LIN {X 0,Y 573.063,Z 619.264,A -85,B 0,C 180,E1 -2090.645,E2 -2090.645} C_VEL
LIN {X 0,Y 573.121,Z 612.909,A -85,B 0,C 180,E1 -2091.584,E2 -2091.584} C_VEL
LIN {X 0,Y 573.201,Z 605.158,A -85,B 0,C 180,E1 -2092.528,E2 -2092.528} C_VEL
LIN {X 0,Y 573.3,Z 596.066,A -85,B 0,C 180,E1 -2093.44,E2 -2093.44} C_VEL
LIN {X 0,Y 573.417,Z 584.971,A -85,B 0,C 180,E1 -2094.337,E2 -2094.337} C_VEL
LIN {X 0,Y 573.555,Z 572.942,A -85,B 0,C 180,E1 -2095.095,E2 -2095.095} C_VEL
LIN {X 0,Y 573.613,Z 562.036,A -85,B 0,C 180,E1 -2095.635,E2 -2095.635} C_VEL
LIN {X 0,Y 573.65,Z 554.886,A -85,B 0,C 180,E1 -2095.926,E2 -2095.926} C_VEL
LIN {X 0,Y 573.305,Z 553.075,A -85,B 0,C 180,E1 -2096.016,E2 -2096.016} C_VEL
LIN {X 0,Y 573.234,Z 553.082,A -85,B 0,C 180,E1 -2098.564,E2 -2098.564} C_VEL
LIN {X 0,Y 573.238,Z 553.081,A -85,B 0,C 180,E1 -2100.992,E2 -2100.992} C_VEL
LIN {X 0,Y 573.256,Z 553.079,A -85,B 0,C 180,E1 -2103.523,E2 -2103.523} C_VEL
LIN {X 0,Y 573.239,Z 553.082,A -85,B 0,C 180,E1 -2106.049,E2 -2106.049} C_VEL
LIN {X 0,Y 573.245,Z 553.083,A -85,B 0,C 180,E1 -2108.7,E2 -2108.7} C_VEL
LIN {X 0,Y 573.305,Z 553.158,A -85,B 0,C 180,E1 -2111.493,E2 -2111.493} C_VEL
LIN {X 0,Y 573.377,Z 559.685,A -85,B 0,C 180,E1 -2113.683,E2 -2113.683} C_VEL
LIN {X 0,Y 573.399,Z 567.264,A -85,B 0,C 180,E1 -2116.313,E2 -2116.313} C_VEL
LIN {X 0,Y 573.383,Z 575.18,A -85,B 0,C 180,E1 -2119.024,E2 -2119.024} C_VEL
LIN {X 0,Y 573.289,Z 582.833,A -85,B 0,C 180,E1 -2121.68,E2 -2121.68} C_VEL
LIN {X 0,Y 573.249,Z 590.784,A -85,B 0,C 180,E1 -2124.414,E2 -2124.414} C_VEL
LIN {X 0,Y 573.184,Z 599.505,A -85,B 0,C 180,E1 -2127.351,E2 -2127.351} C_VEL
LIN {X 0,Y 573.114,Z 608.136,A -85,B 0,C 180,E1 -2130.206,E2 -2130.206} C_VEL
LIN {X 0,Y 573.085,Z 615.536,A -85,B 0,C 180,E1 -2132.621,E2 -2132.621} C_VEL
LIN {X 0,Y 573.073,Z 621.489,A -85,B 0,C 180,E1 -2134.545,E2 -2134.545} C_VEL
LIN {X 0,Y 573.86,Z 627.22,A -85,B 0,C 180,E1 -2134.666,E2 -2134.666} C_VEL
LIN {X 0,Y 573.753,Z 640.519,A -85,B 0,C 180,E1 -2135.015,E2 -2135.015} C_VEL
LIN {X 0,Y 573.656,Z 652.623,A -85,B 0,C 180,E1 -2135.48,E2 -2135.48} C_VEL
LIN {X 0,Y 573.494,Z 663.949,A -85,B 0,C 180,E1 -2136.05,E2 -2136.05} C_VEL
LIN {X 0,Y 573.407,Z 674.306,A -85,B 0,C 180,E1 -2136.708,E2 -2136.708} C_VEL
LIN {X 0,Y 573.316,Z 685.226,A -85,B 0,C 180,E1 -2137.571,E2 -2137.571} C_VEL
LIN {X 0,Y 573.206,Z 693.9,A -85,B 0,C 180,E1 -2138.419,E2 -2138.419} C_VEL
LIN {X 0,Y 573.133,Z 701.824,A -85,B 0,C 180,E1 -2139.357,E2 -2139.357} C_VEL
LIN {X 0,Y 573.082,Z 708.329,A -85,B 0,C 180,E1 -2140.291,E2 -2140.291} C_VEL
LIN {X 0,Y 573.063,Z 714.612,A -85,B 0,C 180,E1 -2141.406,E2 -2141.406} C_VEL
LIN {X 0,Y 572.981,Z 719.505,A -85,B 0,C 180,E1 -2142.512,E2 -2142.512} C_VEL
LIN {X 0,Y 572.958,Z 723.194,A -85,B 0,C 180,E1 -2143.613,E2 -2143.613} C_VEL
LIN {X 0,Y 572.955,Z 725.025,A -85,B 0,C 180,E1 -2144.345,E2 -2144.345} C_VEL
LIN {X 0,Y 572.968,Z 727.243,A -85,B 0,C 180,E1 -2145.694,E2 -2145.694} C_VEL
LIN {X 0,Y 572.962,Z 727.858,A -85,B 0,C 180,E1 -2146.523,E2 -2146.523} C_VEL
LIN {X 0,Y 572.941,Z 727.962,A -85,B 0,C 180,E1 -2147.244,E2 -2147.244} C_VEL
LIN {X 0,Y 572.94,Z 727.643,A -85,B 0,C 180,E1 -2147.964,E2 -2147.964} C_VEL
LIN {X 0,Y 573.025,Z 726.662,A -85,B 0,C 180,E1 -2148.86,E2 -2148.86} C_VEL
LIN {X 0,Y 572.976,Z 724.178,A -85,B 0,C 180,E1 -2150.112,E2 -2150.112} C_VEL
LIN {X 0,Y 572.998,Z 720.982,A -85,B 0,C 180,E1 -2151.181,E2 -2151.181} C_VEL
LIN {X 0,Y 573.046,Z 716.722,A -85,B 0,C 180,E1 -2152.247,E2 -2152.247} C_VEL
LIN {X 0,Y 573.054,Z 710.771,A -85,B 0,C 180,E1 -2153.4,E2 -2153.4} C_VEL
LIN {X 0,Y 573.09,Z 704.512,A -85,B 0,C 180,E1 -2154.37,E2 -2154.37} C_VEL
LIN {X 0,Y 573.163,Z 697.624,A -85,B 0,C 180,E1 -2155.253,E2 -2155.253} C_VEL
LIN {X 0,Y 573.268,Z 689.333,A -85,B 0,C 180,E1 -2156.134,E2 -2156.134} C_VEL
LIN {X 0,Y 573.399,Z 680.335,A -85,B 0,C 180,E1 -2156.926,E2 -2156.926} C_VEL
LIN {X 0,Y 573.463,Z 669.337,A -85,B 0,C 180,E1 -2157.718,E2 -2157.718} C_VEL
LIN {X 0,Y 573.596,Z 656.798,A -85,B 0,C 180,E1 -2158.421,E2 -2158.421} C_VEL
LIN {X 0,Y 573.721,Z 645.415,A -85,B 0,C 180,E1 -2158.904,E2 -2158.904} C_VEL
LIN {X 0,Y 573.801,Z 633.497,A -85,B 0,C 180,E1 -2159.277,E2 -2159.277} C_VEL
LIN {X 0,Y 573.603,Z 624.918,A -85,B 0,C 180,E1 -2159.474,E2 -2159.474} C_VEL
LIN {X 0,Y 573.104,Z 621.456,A -85,B 0,C 180,E1 -2159.561,E2 -2159.561} C_VEL
LIN {X 0,Y 573.138,Z 612.541,A -85,B 0,C 180,E1 -2162.46,E2 -2162.46} C_VEL
LIN {X 0,Y 573.174,Z 603.996,A -85,B 0,C 180,E1 -2165.277,E2 -2165.277} C_VEL
LIN {X 0,Y 573.213,Z 595.549,A -85,B 0,C 180,E1 -2168.106,E2 -2168.106} C_VEL
LIN {X 0,Y 573.281,Z 588.239,A -85,B 0,C 180,E1 -2170.597,E2 -2170.597} C_VEL
LIN {X 0,Y 573.32,Z 579.984,A -85,B 0,C 180,E1 -2173.469,E2 -2173.469} C_VEL
LIN {X 0,Y 573.365,Z 573.728,A -85,B 0,C 180,E1 -2175.645,E2 -2175.645} C_VEL
LIN {X 0,Y 573.328,Z 565.652,A -85,B 0,C 180,E1 -2178.215,E2 -2178.215} C_VEL
LIN {X 0,Y 573.17,Z 557.031,A -85,B 0,C 180,E1 -2180.83,E2 -2180.83} C_VEL
LIN {X 0,Y 573.181,Z 553.092,A -85,B 0,C 180,E1 -2181.961,E2 -2181.961} C_VEL
LIN {X 0,Y 573.264,Z 553.082,A -85,B 0,C 180,E1 -2184.88,E2 -2184.88} C_VEL
LIN {X 0,Y 573.284,Z 553.077,A -85,B 0,C 180,E1 -2187.765,E2 -2187.765} C_VEL
LIN {X 0,Y 573.253,Z 553.083,A -85,B 0,C 180,E1 -2190.176,E2 -2190.176} C_VEL
LIN {X 0,Y 573.253,Z 553.08,A -85,B 0,C 180,E1 -2192.645,E2 -2192.645} C_VEL
LIN {X 0,Y 573.265,Z 553.08,A -85,B 0,C 180,E1 -2195.184,E2 -2195.184} C_VEL
LIN {X 0,Y 573.232,Z 553.083,A -85,B 0,C 180,E1 -2197.808,E2 -2197.808} C_VEL
LIN {X 0,Y 573.265,Z 553.081,A -85,B 0,C 180,E1 -2200.529,E2 -2200.529} C_VEL
LIN {X 0,Y 573.248,Z 553.083,A -85,B 0,C 180,E1 -2203.671,E2 -2203.671} C_VEL
LIN {X 0,Y 573.244,Z 553.083,A -85,B 0,C 180,E1 -2206.643,E2 -2206.643} C_VEL
LIN {X 0,Y 573.271,Z 553.079,A -85,B 0,C 180,E1 -2209.478,E2 -2209.478} C_VEL
LIN {X 0,Y 573.236,Z 553.084,A -85,B 0,C 180,E1 -2212.194,E2 -2212.194} C_VEL
LIN {X 0,Y 573.29,Z 553.151,A -85,B 0,C 180,E1 -2213.301,E2 -2213.301} C_VEL
LIN {X 0,Y 574.101,Z 558.468,A -85,B 0,C 180,E1 -2214.446,E2 -2214.446} C_VEL
LIN {X 0,Y 574.123,Z 573.3,A -85,B 0,C 180,E1 -2217.412,E2 -2217.412} C_VEL
LIN {X 0,Y 574.135,Z 587.619,A -85,B 0,C 180,E1 -2220.163,E2 -2220.163} C_VEL
LIN {X 0,Y 574.037,Z 598.461,A -85,B 0,C 180,E1 -2222.275,E2 -2222.275} C_VEL
LIN {X 0,Y 573.854,Z 614.175,A -85,B 0,C 180,E1 -2225.394,E2 -2225.394} C_VEL
LIN {X 0,Y 573.637,Z 629.889,A -85,B 0,C 180,E1 -2228.436,E2 -2228.436} C_VEL
LIN {X 0,Y 573.459,Z 645.603,A -85,B 0,C 180,E1 -2231.42,E2 -2231.42} C_VEL
LIN {X 0,Y 573.327,Z 659.353,A -85,B 0,C 180,E1 -2233.99,E2 -2233.99} C_VEL
LIN {X 0,Y 573.205,Z 675.067,A -85,B 0,C 180,E1 -2236.89,E2 -2236.89} C_VEL
LIN {X 0,Y 573.204,Z 678.139,A -85,B 0,C 180,E1 -2237.453,E2 -2237.453} C_VEL
LIN {X 0,Y 573.867,Z 683.985,A -85,B 0,C 180,E1 -2237.558,E2 -2237.558} C_VEL
LIN {X 0,Y 573.787,Z 697.245,A -85,B 0,C 180,E1 -2237.87,E2 -2237.87} C_VEL
LIN {X 0,Y 573.713,Z 709.391,A -85,B 0,C 180,E1 -2238.295,E2 -2238.295} C_VEL
LIN {X 0,Y 573.573,Z 720.61,A -85,B 0,C 180,E1 -2238.818,E2 -2238.818} C_VEL
LIN {X 0,Y 573.471,Z 731.924,A -85,B 0,C 180,E1 -2239.497,E2 -2239.497} C_VEL
LIN {X 0,Y 573.351,Z 742.548,A -85,B 0,C 180,E1 -2240.298,E2 -2240.298} C_VEL
LIN {X 0,Y 573.24,Z 752.12,A -85,B 0,C 180,E1 -2241.185,E2 -2241.185} C_VEL
LIN {X 0,Y 573.16,Z 759.966,A -85,B 0,C 180,E1 -2242.072,E2 -2242.072} C_VEL
LIN {X 0,Y 573.072,Z 767.958,A -85,B 0,C 180,E1 -2243.186,E2 -2243.186} C_VEL
LIN {X 0,Y 573.07,Z 774.684,A -85,B 0,C 180,E1 -2244.37,E2 -2244.37} C_VEL
LIN {X 0,Y 573.029,Z 779.374,A -85,B 0,C 180,E1 -2245.428,E2 -2245.428} C_VEL
LIN {X 0,Y 573.022,Z 782.959,A -85,B 0,C 180,E1 -2246.485,E2 -2246.485} C_VEL
LIN {X 0,Y 572.959,Z 784.81,A -85,B 0,C 180,E1 -2247.188,E2 -2247.188} C_VEL
LIN {X 0,Y 572.937,Z 786.201,A -85,B 0,C 180,E1 -2247.892,E2 -2247.892} C_VEL
LIN {X 0,Y 572.94,Z 787.785,A -85,B 0,C 180,E1 -2249.298,E2 -2249.298} C_VEL
LIN {X 0,Y 572.938,Z 788,A -85,B 0,C 180,E1 -2250.001,E2 -2250.001} C_VEL
LIN {X 0,Y 572.946,Z 787.185,A -85,B 0,C 180,E1 -2251.406,E2 -2251.406} C_VEL
LIN {X 0,Y 572.937,Z 786.199,A -85,B 0,C 180,E1 -2252.11,E2 -2252.11} C_VEL
LIN {X 0,Y 572.959,Z 784.808,A -85,B 0,C 180,E1 -2252.813,E2 -2252.813} C_VEL
LIN {X 0,Y 573.014,Z 781.894,A -85,B 0,C 180,E1 -2253.869,E2 -2253.869} C_VEL
LIN {X 0,Y 572.963,Z 777.947,A -85,B 0,C 180,E1 -2254.926,E2 -2254.926} C_VEL
LIN {X 0,Y 573.064,Z 771.874,A -85,B 0,C 180,E1 -2256.161,E2 -2256.161} C_VEL
LIN {X 0,Y 573.12,Z 765.233,A -85,B 0,C 180,E1 -2257.221,E2 -2257.221} C_VEL
LIN {X 0,Y 573.199,Z 756.985,A -85,B 0,C 180,E1 -2258.284,E2 -2258.284} C_VEL
LIN {X 0,Y 573.287,Z 748.532,A -85,B 0,C 180,E1 -2259.171,E2 -2259.171} C_VEL
LIN {X 0,Y 573.42,Z 738.089,A -85,B 0,C 180,E1 -2260.059,E2 -2260.059} C_VEL
LIN {X 0,Y 573.554,Z 726.423,A -85,B 0,C 180,E1 -2260.853,E2 -2260.853} C_VEL
LIN {X 0,Y 573.618,Z 714.869,A -85,B 0,C 180,E1 -2261.467,E2 -2261.467} C_VEL
LIN {X 0,Y 573.731,Z 702.158,A -85,B 0,C 180,E1 -2261.975,E2 -2261.975} C_VEL
LIN {X 0,Y 573.855,Z 689.497,A -85,B 0,C 180,E1 -2262.331,E2 -2262.331} C_VEL
LIN {X 0,Y 573.668,Z 681.259,A -85,B 0,C 180,E1 -2262.49,E2 -2262.49} C_VEL
LIN {X 0,Y 573.194,Z 678.031,A -85,B 0,C 180,E1 -2262.571,E2 -2262.571} C_VEL
LIN {X 0,Y 573.319,Z 663.358,A -85,B 0,C 180,E1 -2265.282,E2 -2265.282} C_VEL
LIN {X 0,Y 573.458,Z 647.707,A -85,B 0,C 180,E1 -2268.211,E2 -2268.211} C_VEL
LIN {X 0,Y 573.616,Z 632.538,A -85,B 0,C 180,E1 -2271.096,E2 -2271.096} C_VEL
LIN {X 0,Y 573.768,Z 618.361,A -85,B 0,C 180,E1 -2273.842,E2 -2273.842} C_VEL
LIN {X 0,Y 573.962,Z 604.222,A -85,B 0,C 180,E1 -2276.637,E2 -2276.637} C_VEL
LIN {X 0,Y 574.103,Z 590.754,A -85,B 0,C 180,E1 -2279.319,E2 -2279.319} C_VEL
LIN {X 0,Y 574.085,Z 576.51,A -85,B 0,C 180,E1 -2282.063,E2 -2282.063} C_VEL
LIN {X 0,Y 574.126,Z 563.882,A -85,B 0,C 180,E1 -2284.583,E2 -2284.583} C_VEL
LIN {X 0,Y 573.987,Z 556.687,A -85,B 0,C 180,E1 -2286.087,E2 -2286.087} C_VEL
LIN {X 0,Y 573.258,Z 553.081,A -85,B 0,C 180,E1 -2286.922,E2 -2286.922} C_VEL
LIN {X 0,Y 573.253,Z 553.082,A -85,B 0,C 180,E1 -2289.607,E2 -2289.607} C_VEL
LIN {X 0,Y 573.245,Z 553.08,A -85,B 0,C 180,E1 -2292.642,E2 -2292.642} C_VEL
LIN {X 0,Y 573.237,Z 553.084,A -85,B 0,C 180,E1 -2295.666,E2 -2295.666} C_VEL
LIN {X 0,Y 573.243,Z 553.081,A -85,B 0,C 180,E1 -2298.544,E2 -2298.544} C_VEL
LIN {X 0,Y 573.243,Z 553.082,A -85,B 0,C 180,E1 -2301.298,E2 -2301.298} C_VEL
LIN {X 0,Y 573.27,Z 553.079,A -85,B 0,C 180,E1 -2304.011,E2 -2304.011} C_VEL
LIN {X 0,Y 573.274,Z 553.077,A -85,B 0,C 180,E1 -2306.518,E2 -2306.518} C_VEL
LIN {X 0,Y 573.232,Z 553.082,A -85,B 0,C 180,E1 -2309.118,E2 -2309.118} C_VEL
LIN {X 0,Y 573.268,Z 553.08,A -85,B 0,C 180,E1 -2311.969,E2 -2311.969} C_VEL
LIN {X 0,Y 573.259,Z 553.079,A -85,B 0,C 180,E1 -2314.59,E2 -2314.59} C_VEL
LIN {X 0,Y 573.241,Z 553.082,A -85,B 0,C 180,E1 -2317.662,E2 -2317.662} C_VEL
LIN {X 0,Y 573.283,Z 553.076,A -85,B 0,C 180,E1 -2320.728,E2 -2320.728} C_VEL
LIN {X 0,Y 573.256,Z 553.081,A -85,B 0,C 180,E1 -2323.622,E2 -2323.622} C_VEL
LIN {X 0,Y 573.277,Z 553.077,A -85,B 0,C 180,E1 -2325.807,E2 -2325.807} C_VEL
LIN {X 0,Y 573.267,Z 553.078,A -85,B 0,C 180,E1 -2328.745,E2 -2328.745} C_VEL
LIN {X 0,Y 573.293,Z 553.075,A -85,B 0,C 180,E1 -2331.54,E2 -2331.54} C_VEL
LIN {X 0,Y 573.294,Z 553.076,A -85,B 0,C 180,E1 -2334.372,E2 -2334.372} C_VEL
LIN {X 0,Y 573.306,Z 553.074,A -85,B 0,C 180,E1 -2337.892,E2 -2337.892} C_VEL
LIN {X 0,Y 573.336,Z 553.069,A -85,B 0,C 180,E1 -2340.702,E2 -2340.702} C_VEL
LIN {X 0,Y 573.233,Z 553.084,A -85,B 0,C 180,E1 -2343.514,E2 -2343.514} C_VEL
LIN {X 0,Y 573.293,Z 553.075,A -85,B 0,C 180,E1 -2345.628,E2 -2345.628} C_VEL
LIN {X 0,Y 573.288,Z 553.076,A -85,B 0,C 180,E1 -2348.459,E2 -2348.459} C_VEL
LIN {X 0,Y 573.275,Z 553.077,A -85,B 0,C 180,E1 -2351.312,E2 -2351.312} C_VEL
LIN {X 0,Y 573.277,Z 553.078,A -85,B 0,C 180,E1 -2354.193,E2 -2354.193} C_VEL
LIN {X 0,Y 573.261,Z 553.079,A -85,B 0,C 180,E1 -2357.111,E2 -2357.111} C_VEL
LIN {X 0,Y 573.254,Z 553.081,A -85,B 0,C 180,E1 -2360.076,E2 -2360.076} C_VEL
LIN {X 0,Y 573.237,Z 553.082,A -85,B 0,C 180,E1 -2363.099,E2 -2363.099} C_VEL
LIN {X 0,Y 573.252,Z 553.079,A -85,B 0,C 180,E1 -2364.389,E2 -2364.389} C_VEL
LIN {X 0,Y 572.624,Z 553.16,A -85,B 0,C 180,E1 -2364.975,E2 -2364.975} C_VEL
LIN {X 0,Y 569.777,Z 553.515,A -85,B 0,C 180,E1 -2365.927,E2 -2365.927} C_VEL
LIN {X 0,Y 567.345,Z 553.817,A -85,B 0,C 180,E1 -2366.692,E2 -2366.692} C_VEL
LIN {X 0,Y 566.295,Z 553.945,A -85,B 0,C 180,E1 -2367.283,E2 -2367.283} C_VEL
LIN {X 0,Y 566.209,Z 553.956,A -85,B 0,C 180,E1 -2367.483,E2 -2367.483} C_VEL
LIN {X 0,Y 566.203,Z 553.957,A -85,B 0,C 180,E1 -2369.768,E2 -2369.768} C_VEL
LIN {X 0,Y 566.205,Z 553.958,A -85,B 0,C 180,E1 -2372.43,E2 -2372.43} C_VEL
LIN {X 0,Y 566.214,Z 553.959,A -85,B 0,C 180,E1 -2374.994,E2 -2374.994} C_VEL
LIN {X 0,Y 566.198,Z 553.96,A -85,B 0,C 180,E1 -2377.46,E2 -2377.46} C_VEL
LIN {X 0,Y 566.219,Z 553.956,A -85,B 0,C 180,E1 -2380.198,E2 -2380.198} C_VEL
LIN {X 0,Y 566.206,Z 553.959,A -85,B 0,C 180,E1 -2383.053,E2 -2383.053} C_VEL
LIN {X 0,Y 566.203,Z 553.958,A -85,B 0,C 180,E1 -2386.048,E2 -2386.048} C_VEL
LIN {X 0,Y 566.213,Z 553.958,A -85,B 0,C 180,E1 -2388.863,E2 -2388.863} C_VEL
LIN {X 0,Y 566.191,Z 553.96,A -85,B 0,C 180,E1 -2391.637,E2 -2391.637} C_VEL
LIN {X 0,Y 566.163,Z 553.963,A -85,B 0,C 180,E1 -2394.307,E2 -2394.307} C_VEL
LIN {X 0,Y 566.222,Z 553.956,A -85,B 0,C 180,E1 -2396.897,E2 -2396.897} C_VEL
LIN {X 0,Y 566.19,Z 553.961,A -85,B 0,C 180,E1 -2399.407,E2 -2399.407} C_VEL
LIN {X 0,Y 566.212,Z 553.958,A -85,B 0,C 180,E1 -2401.857,E2 -2401.857} C_VEL
LIN {X 0,Y 566.217,Z 553.959,A -85,B 0,C 180,E1 -2404.251,E2 -2404.251} C_VEL
LIN {X 0,Y 566.193,Z 553.961,A -85,B 0,C 180,E1 -2406.713,E2 -2406.713} C_VEL
LIN {X 0,Y 566.213,Z 553.956,A -85,B 0,C 180,E1 -2409.662,E2 -2409.662} C_VEL
LIN {X 0,Y 566.2,Z 553.959,A -85,B 0,C 180,E1 -2412.668,E2 -2412.668} C_VEL
LIN {X 0,Y 566.234,Z 553.954,A -85,B 0,C 180,E1 -2415.626,E2 -2415.626} C_VEL
LIN {X 0,Y 566.235,Z 553.954,A -85,B 0,C 180,E1 -2418.674,E2 -2418.674} C_VEL
LIN {X 0,Y 566.228,Z 553.955,A -85,B 0,C 180,E1 -2421.434,E2 -2421.434} C_VEL
LIN {X 0,Y 566.259,Z 553.952,A -85,B 0,C 180,E1 -2424.301,E2 -2424.301} C_VEL
LIN {X 0,Y 566.284,Z 553.949,A -85,B 0,C 180,E1 -2427.866,E2 -2427.866} C_VEL
LIN {X 0,Y 566.299,Z 553.946,A -85,B 0,C 180,E1 -2430.71,E2 -2430.71} C_VEL
LIN {X 0,Y 566.275,Z 554.004,A -85,B 0,C 180,E1 -2431.977,E2 -2431.977} C_VEL
LIN {X 0,Y 566.733,Z 557.867,A -85,B 0,C 180,E1 -2432.131,E2 -2432.131} C_VEL
LIN {X 0,Y 566.607,Z 569.41,A -85,B 0,C 180,E1 -2432.665,E2 -2432.665} C_VEL
LIN {X 0,Y 566.525,Z 578.649,A -85,B 0,C 180,E1 -2433.199,E2 -2433.199} C_VEL
LIN {X 0,Y 566.351,Z 588.706,A -85,B 0,C 180,E1 -2433.913,E2 -2433.913} C_VEL
LIN {X 0,Y 566.246,Z 597.047,A -85,B 0,C 180,E1 -2434.627,E2 -2434.627} C_VEL
LIN {X 0,Y 566.182,Z 604.132,A -85,B 0,C 180,E1 -2435.341,E2 -2435.341} C_VEL
LIN {X 0,Y 566.126,Z 611.583,A -85,B 0,C 180,E1 -2436.235,E2 -2436.235} C_VEL
LIN {X 0,Y 566.053,Z 617.821,A -85,B 0,C 180,E1 -2437.131,E2 -2437.131} C_VEL
LIN {X 0,Y 565.982,Z 622.123,A -85,B 0,C 180,E1 -2437.85,E2 -2437.85} C_VEL
LIN {X 0,Y 565.941,Z 627.374,A -85,B 0,C 180,E1 -2438.929,E2 -2438.929} C_VEL
LIN {X 0,Y 565.925,Z 631.479,A -85,B 0,C 180,E1 -2440.012,E2 -2440.012} C_VEL
LIN {X 0,Y 565.882,Z 634.643,A -85,B 0,C 180,E1 -2441.146,E2 -2441.146} C_VEL
LIN {X 0,Y 565.863,Z 636.61,A -85,B 0,C 180,E1 -2442.188,E2 -2442.188} C_VEL
LIN {X 0,Y 565.842,Z 637.503,A -85,B 0,C 180,E1 -2442.918,E2 -2442.918} C_VEL
LIN {X 0,Y 565.872,Z 637.914,A -85,B 0,C 180,E1 -2444.382,E2 -2444.382} C_VEL
LIN {X 0,Y 565.809,Z 637.547,A -85,B 0,C 180,E1 -2445.119,E2 -2445.119} C_VEL
LIN {X 0,Y 565.87,Z 635.393,A -85,B 0,C 180,E1 -2446.597,E2 -2446.597} C_VEL
LIN {X 0,Y 565.898,Z 632.603,A -85,B 0,C 180,E1 -2447.713,E2 -2447.713} C_VEL
LIN {X 0,Y 565.905,Z 628.683,A -85,B 0,C 180,E1 -2448.837,E2 -2448.837} C_VEL
LIN {X 0,Y 565.965,Z 625.43,A -85,B 0,C 180,E1 -2449.589,E2 -2449.589} C_VEL
LIN {X 0,Y 566,Z 619.275,A -85,B 0,C 180,E1 -2450.724,E2 -2450.724} C_VEL
LIN {X 0,Y 566.078,Z 612.656,A -85,B 0,C 180,E1 -2451.711,E2 -2451.711} C_VEL
LIN {X 0,Y 566.15,Z 605.171,A -85,B 0,C 180,E1 -2452.632,E2 -2452.632} C_VEL
LIN {X 0,Y 566.26,Z 596.693,A -85,B 0,C 180,E1 -2453.497,E2 -2453.497} C_VEL
LIN {X 0,Y 566.375,Z 586.308,A -85,B 0,C 180,E1 -2454.367,E2 -2454.367} C_VEL
LIN {X 0,Y 566.561,Z 575.227,A -85,B 0,C 180,E1 -2455.105,E2 -2455.105} C_VEL
LIN {X 0,Y 566.628,Z 563.2,A -85,B 0,C 180,E1 -2455.728,E2 -2455.728} C_VEL
LIN {X 0,Y 566.545,Z 555.337,A -85,B 0,C 180,E1 -2456.061,E2 -2456.061} C_VEL
LIN {X 0,Y 566.248,Z 553.953,A -85,B 0,C 180,E1 -2456.117,E2 -2456.117} C_VEL
LIN {X 0,Y 566.19,Z 553.96,A -85,B 0,C 180,E1 -2458.952,E2 -2458.952} C_VEL
LIN {X 0,Y 566.2,Z 553.959,A -85,B 0,C 180,E1 -2461.42,E2 -2461.42} C_VEL
LIN {X 0,Y 566.204,Z 553.959,A -85,B 0,C 180,E1 -2463.955,E2 -2463.955} C_VEL
LIN {X 0,Y 566.205,Z 553.958,A -85,B 0,C 180,E1 -2466.568,E2 -2466.568} C_VEL
LIN {X 0,Y 566.21,Z 553.959,A -85,B 0,C 180,E1 -2469.686,E2 -2469.686} C_VEL
LIN {X 0,Y 566.259,Z 554.067,A -85,B 0,C 180,E1 -2471.427,E2 -2471.427} C_VEL
LIN {X 0,Y 566.367,Z 561.664,A -85,B 0,C 180,E1 -2474.018,E2 -2474.018} C_VEL
LIN {X 0,Y 566.354,Z 570.107,A -85,B 0,C 180,E1 -2476.961,E2 -2476.961} C_VEL
LIN {X 0,Y 566.313,Z 578.345,A -85,B 0,C 180,E1 -2479.81,E2 -2479.81} C_VEL
LIN {X 0,Y 566.246,Z 586.39,A -85,B 0,C 180,E1 -2482.591,E2 -2482.591} C_VEL
LIN {X 0,Y 566.192,Z 593.88,A -85,B 0,C 180,E1 -2485.181,E2 -2485.181} C_VEL
LIN {X 0,Y 566.104,Z 602.65,A -85,B 0,C 180,E1 -2488.155,E2 -2488.155} C_VEL
LIN {X 0,Y 566.055,Z 610.261,A -85,B 0,C 180,E1 -2490.695,E2 -2490.695} C_VEL
LIN {X 0,Y 566.004,Z 618.62,A -85,B 0,C 180,E1 -2493.448,E2 -2493.448} C_VEL
LIN {X 0,Y 566.002,Z 621.485,A -85,B 0,C 180,E1 -2494.385,E2 -2494.385} C_VEL
LIN {X 0,Y 566.933,Z 628.252,A -85,B 0,C 180,E1 -2494.533,E2 -2494.533} C_VEL
LIN {X 0,Y 566.807,Z 640.989,A -85,B 0,C 180,E1 -2494.882,E2 -2494.882} C_VEL
LIN {X 0,Y 566.684,Z 651.94,A -85,B 0,C 180,E1 -2495.305,E2 -2495.305} C_VEL
LIN {X 0,Y 566.562,Z 662.569,A -85,B 0,C 180,E1 -2495.836,E2 -2495.836} C_VEL
LIN {X 0,Y 566.415,Z 673.305,A -85,B 0,C 180,E1 -2496.509,E2 -2496.509} C_VEL
LIN {X 0,Y 566.314,Z 683.208,A -85,B 0,C 180,E1 -2497.278,E2 -2497.278} C_VEL
LIN {X 0,Y 566.188,Z 693.661,A -85,B 0,C 180,E1 -2498.285,E2 -2498.285} C_VEL
LIN {X 0,Y 566.072,Z 701.953,A -85,B 0,C 180,E1 -2499.278,E2 -2499.278} C_VEL
LIN {X 0,Y 566.014,Z 708.432,A -85,B 0,C 180,E1 -2500.224,E2 -2500.224} C_VEL
LIN {X 0,Y 565.975,Z 713.754,A -85,B 0,C 180,E1 -2501.165,E2 -2501.165} C_VEL
LIN {X 0,Y 565.909,Z 718.829,A -85,B 0,C 180,E1 -2502.286,E2 -2502.286} C_VEL
LIN {X 0,Y 565.878,Z 722.693,A -85,B 0,C 180,E1 -2503.402,E2 -2503.402} C_VEL
LIN {X 0,Y 565.849,Z 724.661,A -85,B 0,C 180,E1 -2504.143,E2 -2504.143} C_VEL
LIN {X 0,Y 565.834,Z 726.163,A -85,B 0,C 180,E1 -2504.881,E2 -2504.881} C_VEL
LIN {X 0,Y 565.873,Z 727.192,A -85,B 0,C 180,E1 -2505.632,E2 -2505.632} C_VEL
LIN {X 0,Y 565.839,Z 727.997,A -85,B 0,C 180,E1 -2507.082,E2 -2507.082} C_VEL
LIN {X 0,Y 565.859,Z 727.749,A -85,B 0,C 180,E1 -2507.811,E2 -2507.811} C_VEL
LIN {X 0,Y 565.907,Z 726.071,A -85,B 0,C 180,E1 -2509.264,E2 -2509.264} C_VEL
LIN {X 0,Y 565.902,Z 724.574,A -85,B 0,C 180,E1 -2509.988,E2 -2509.988} C_VEL
LIN {X 0,Y 565.912,Z 720.3,A -85,B 0,C 180,E1 -2511.43,E2 -2511.43} C_VEL
LIN {X 0,Y 565.962,Z 715.83,A -85,B 0,C 180,E1 -2512.508,E2 -2512.508} C_VEL
LIN {X 0,Y 565.965,Z 710.152,A -85,B 0,C 180,E1 -2513.584,E2 -2513.584} C_VEL
LIN {X 0,Y 566.007,Z 704.39,A -85,B 0,C 180,E1 -2514.478,E2 -2514.478} C_VEL
LIN {X 0,Y 566.108,Z 697.476,A -85,B 0,C 180,E1 -2515.372,E2 -2515.372} C_VEL
LIN {X 0,Y 566.229,Z 689.159,A -85,B 0,C 180,E1 -2516.264,E2 -2516.264} C_VEL
LIN {X 0,Y 566.361,Z 680.134,A -85,B 0,C 180,E1 -2517.066,E2 -2517.066} C_VEL
LIN {X 0,Y 566.476,Z 669.084,A -85,B 0,C 180,E1 -2517.867,E2 -2517.867} C_VEL
LIN {X 0,Y 566.63,Z 656.431,A -85,B 0,C 180,E1 -2518.579,E2 -2518.579} C_VEL
LIN {X 0,Y 566.77,Z 644.936,A -85,B 0,C 180,E1 -2519.068,E2 -2519.068} C_VEL
LIN {X 0,Y 566.885,Z 632.821,A -85,B 0,C 180,E1 -2519.445,E2 -2519.445} C_VEL
LIN {X 0,Y 566.662,Z 625.829,A -85,B 0,C 180,E1 -2519.612,E2 -2519.612} C_VEL
LIN {X 0,Y 566.048,Z 621.482,A -85,B 0,C 180,E1 -2519.711,E2 -2519.711} C_VEL
LIN {X 0,Y 566.078,Z 613.043,A -85,B 0,C 180,E1 -2522.491,E2 -2522.491} C_VEL
LIN {X 0,Y 566.12,Z 604.499,A -85,B 0,C 180,E1 -2525.343,E2 -2525.343} C_VEL
LIN {X 0,Y 566.181,Z 596.054,A -85,B 0,C 180,E1 -2528.207,E2 -2528.207} C_VEL
LIN {X 0,Y 566.27,Z 586.978,A -85,B 0,C 180,E1 -2531.347,E2 -2531.347} C_VEL
LIN {X 0,Y 566.322,Z 579.399,A -85,B 0,C 180,E1 -2534.004,E2 -2534.004} C_VEL
LIN {X 0,Y 566.319,Z 573.899,A -85,B 0,C 180,E1 -2535.844,E2 -2535.844} C_VEL
LIN {X 0,Y 566.261,Z 565.699,A -85,B 0,C 180,E1 -2538.451,E2 -2538.451} C_VEL
LIN {X 0,Y 566.147,Z 556.905,A -85,B 0,C 180,E1 -2541.1,E2 -2541.1} C_VEL
LIN {X 0,Y 566.126,Z 553.97,A -85,B 0,C 180,E1 -2541.961,E2 -2541.961} C_VEL
LIN {X 0,Y 566.194,Z 553.961,A -85,B 0,C 180,E1 -2544.181,E2 -2544.181} C_VEL
LIN {X 0,Y 566.231,Z 553.955,A -85,B 0,C 180,E1 -2546.666,E2 -2546.666} C_VEL
LIN {X 0,Y 566.224,Z 553.956,A -85,B 0,C 180,E1 -2549.678,E2 -2549.678} C_VEL
LIN {X 0,Y 566.205,Z 553.959,A -85,B 0,C 180,E1 -2552.432,E2 -2552.432} C_VEL
LIN {X 0,Y 566.21,Z 553.958,A -85,B 0,C 180,E1 -2554.996,E2 -2554.996} C_VEL
LIN {X 0,Y 566.192,Z 553.962,A -85,B 0,C 180,E1 -2557.462,E2 -2557.462} C_VEL
LIN {X 0,Y 566.223,Z 553.956,A -85,B 0,C 180,E1 -2560.198,E2 -2560.198} C_VEL
LIN {X 0,Y 566.201,Z 553.958,A -85,B 0,C 180,E1 -2563.055,E2 -2563.055} C_VEL
LIN {X 0,Y 566.199,Z 553.959,A -85,B 0,C 180,E1 -2566.049,E2 -2566.049} C_VEL
LIN {X 0,Y 566.209,Z 553.96,A -85,B 0,C 180,E1 -2568.865,E2 -2568.865} C_VEL
LIN {X 0,Y 566.189,Z 553.962,A -85,B 0,C 180,E1 -2571.638,E2 -2571.638} C_VEL
LIN {X 0,Y 566.248,Z 554.083,A -85,B 0,C 180,E1 -2573.102,E2 -2573.102} C_VEL
LIN {X 0,Y 567.188,Z 559.929,A -85,B 0,C 180,E1 -2574.383,E2 -2574.383} C_VEL
LIN {X 0,Y 567.181,Z 573.961,A -85,B 0,C 180,E1 -2577.233,E2 -2577.233} C_VEL
LIN {X 0,Y 567.148,Z 589.042,A -85,B 0,C 180,E1 -2580.162,E2 -2580.162} C_VEL
LIN {X 0,Y 567.077,Z 603.796,A -85,B 0,C 180,E1 -2582.993,E2 -2582.993} C_VEL
LIN {X 0,Y 566.839,Z 618.103,A -85,B 0,C 180,E1 -2585.849,E2 -2585.849} C_VEL
LIN {X 0,Y 566.632,Z 632.656,A -85,B 0,C 180,E1 -2588.694,E2 -2588.694} C_VEL
LIN {X 0,Y 566.455,Z 647.567,A -85,B 0,C 180,E1 -2591.557,E2 -2591.557} C_VEL
LIN {X 0,Y 566.286,Z 663.281,A -85,B 0,C 180,E1 -2594.525,E2 -2594.525} C_VEL
LIN {X 0,Y 566.157,Z 678.141,A -85,B 0,C 180,E1 -2597.295,E2 -2597.295} C_VEL
LIN {X 0,Y 566.964,Z 685.127,A -85,B 0,C 180,E1 -2597.427,E2 -2597.427} C_VEL
LIN {X 0,Y 566.825,Z 698.765,A -85,B 0,C 180,E1 -2597.765,E2 -2597.765} C_VEL
LIN {X 0,Y 566.719,Z 711.541,A -85,B 0,C 180,E1 -2598.239,E2 -2598.239} C_VEL
LIN {X 0,Y 566.566,Z 723.855,A -85,B 0,C 180,E1 -2598.861,E2 -2598.861} C_VEL
LIN {X 0,Y 566.419,Z 734.491,A -85,B 0,C 180,E1 -2599.546,E2 -2599.546} C_VEL
LIN {X 0,Y 566.3,Z 744.655,A -85,B 0,C 180,E1 -2600.356,E2 -2600.356} C_VEL
LIN {X 0,Y 566.166,Z 753.793,A -85,B 0,C 180,E1 -2601.254,E2 -2601.254} C_VEL
LIN {X 0,Y 566.08,Z 762.695,A -85,B 0,C 180,E1 -2602.331,E2 -2602.331} C_VEL
LIN {X 0,Y 565.967,Z 769.96,A -85,B 0,C 180,E1 -2603.423,E2 -2603.423} C_VEL
LIN {X 0,Y 566.004,Z 774.684,A -85,B 0,C 180,E1 -2604.3,E2 -2604.3} C_VEL
LIN {X 0,Y 565.933,Z 779.375,A -85,B 0,C 180,E1 -2605.371,E2 -2605.371} C_VEL
LIN {X 0,Y 565.927,Z 782.959,A -85,B 0,C 180,E1 -2606.441,E2 -2606.441} C_VEL
LIN {X 0,Y 565.878,Z 784.81,A -85,B 0,C 180,E1 -2607.153,E2 -2607.153} C_VEL
LIN {X 0,Y 565.846,Z 787.186,A -85,B 0,C 180,E1 -2608.577,E2 -2608.577} C_VEL
LIN {X 0,Y 565.839,Z 788,A -85,B 0,C 180,E1 -2610.001,E2 -2610.001} C_VEL
LIN {X 0,Y 565.846,Z 787.185,A -85,B 0,C 180,E1 -2611.424,E2 -2611.424} C_VEL
LIN {X 0,Y 565.838,Z 786.199,A -85,B 0,C 180,E1 -2612.136,E2 -2612.136} C_VEL
LIN {X 0,Y 565.878,Z 784.808,A -85,B 0,C 180,E1 -2612.848,E2 -2612.848} C_VEL
LIN {X 0,Y 565.926,Z 781.894,A -85,B 0,C 180,E1 -2613.917,E2 -2613.917} C_VEL
LIN {X 0,Y 565.878,Z 777.947,A -85,B 0,C 180,E1 -2614.988,E2 -2614.988} C_VEL
LIN {X 0,Y 566.002,Z 772.863,A -85,B 0,C 180,E1 -2616.059,E2 -2616.059} C_VEL
LIN {X 0,Y 566.041,Z 766.465,A -85,B 0,C 180,E1 -2617.133,E2 -2617.133} C_VEL
LIN {X 0,Y 566.133,Z 758.473,A -85,B 0,C 180,E1 -2618.208,E2 -2618.208} C_VEL
LIN {X 0,Y 566.229,Z 750.33,A -85,B 0,C 180,E1 -2619.106,E2 -2619.106} C_VEL
LIN {X 0,Y 566.341,Z 740.394,A -85,B 0,C 180,E1 -2620.006,E2 -2620.006} C_VEL
LIN {X 0,Y 566.511,Z 729.298,A -85,B 0,C 180,E1 -2620.807,E2 -2620.807} C_VEL
LIN {X 0,Y 566.614,Z 718.167,A -85,B 0,C 180,E1 -2621.447,E2 -2621.447} C_VEL
LIN {X 0,Y 566.768,Z 705.972,A -85,B 0,C 180,E1 -2621.988,E2 -2621.988} C_VEL
LIN {X 0,Y 566.888,Z 693.154,A -85,B 0,C 180,E1 -2622.394,E2 -2622.394} C_VEL
LIN {X 0,Y 566.749,Z 682.03,A -85,B 0,C 180,E1 -2622.633,E2 -2622.633} C_VEL
LIN {X 0,Y 566.156,Z 678.031,A -85,B 0,C 180,E1 -2622.73,E2 -2622.73} C_VEL
LIN {X 0,Y 566.288,Z 663.358,A -85,B 0,C 180,E1 -2625.476,E2 -2625.476} C_VEL
LIN {X 0,Y 566.43,Z 649.663,A -85,B 0,C 180,E1 -2628.071,E2 -2628.071} C_VEL
LIN {X 0,Y 566.617,Z 634.012,A -85,B 0,C 180,E1 -2631.082,E2 -2631.082} C_VEL
LIN {X 0,Y 566.808,Z 620.319,A -85,B 0,C 180,E1 -2633.764,E2 -2633.764} C_VEL
LIN {X 0,Y 567.03,Z 606.622,A -85,B 0,C 180,E1 -2636.501,E2 -2636.501} C_VEL
LIN {X 0,Y 567.112,Z 594.35,A -85,B 0,C 180,E1 -2638.902,E2 -2638.902} C_VEL
LIN {X 0,Y 567.155,Z 580.607,A -85,B 0,C 180,E1 -2641.571,E2 -2641.571} C_VEL
LIN {X 0,Y 567.17,Z 567.981,A -85,B 0,C 180,E1 -2644.105,E2 -2644.105} C_VEL
LIN {X 0,Y 567.181,Z 559.117,A -85,B 0,C 180,E1 -2645.955,E2 -2645.955} C_VEL
LIN {X 0,Y 566.215,Z 553.959,A -85,B 0,C 180,E1 -2647.125,E2 -2647.125} C_VEL
LIN {X 0,Y 566.217,Z 553.959,A -85,B 0,C 180,E1 -2649.686,E2 -2649.686} C_VEL
LIN {X 0,Y 566.218,Z 553.959,A -85,B 0,C 180,E1 -2652.087,E2 -2652.087} C_VEL
LIN {X 0,Y 566.178,Z 553.961,A -85,B 0,C 180,E1 -2655.036,E2 -2655.036} C_VEL
LIN {X 0,Y 566.216,Z 553.959,A -85,B 0,C 180,E1 -2657.913,E2 -2657.913} C_VEL
LIN {X 0,Y 566.217,Z 553.956,A -85,B 0,C 180,E1 -2660.726,E2 -2660.726} C_VEL
LIN {X 0,Y 566.223,Z 553.958,A -85,B 0,C 180,E1 -2663.783,E2 -2663.783} C_VEL
LIN {X 0,Y 566.217,Z 553.958,A -85,B 0,C 180,E1 -2666.266,E2 -2666.266} C_VEL
LIN {X 0,Y 566.194,Z 553.958,A -85,B 0,C 180,E1 -2668.924,E2 -2668.924} C_VEL
LIN {X 0,Y 566.234,Z 553.955,A -85,B 0,C 180,E1 -2671.858,E2 -2671.858} C_VEL
LIN {X 0,Y 566.219,Z 553.958,A -85,B 0,C 180,E1 -2674.251,E2 -2674.251} C_VEL
LIN {X 0,Y 566.177,Z 553.963,A -85,B 0,C 180,E1 -2676.718,E2 -2676.718} C_VEL
LIN {X 0,Y 566.218,Z 553.955,A -85,B 0,C 180,E1 -2679.663,E2 -2679.663} C_VEL
LIN {X 0,Y 566.203,Z 553.959,A -85,B 0,C 180,E1 -2682.668,E2 -2682.668} C_VEL
LIN {X 0,Y 566.238,Z 553.953,A -85,B 0,C 180,E1 -2685.627,E2 -2685.627} C_VEL
LIN {X 0,Y 566.239,Z 553.953,A -85,B 0,C 180,E1 -2688.675,E2 -2688.675} C_VEL
LIN {X 0,Y 566.237,Z 553.953,A -85,B 0,C 180,E1 -2691.434,E2 -2691.434} C_VEL
LIN {X 0,Y 566.263,Z 553.952,A -85,B 0,C 180,E1 -2694.301,E2 -2694.301} C_VEL
LIN {X 0,Y 566.278,Z 553.95,A -85,B 0,C 180,E1 -2697.866,E2 -2697.866} C_VEL
LIN {X 0,Y 566.307,Z 553.945,A -85,B 0,C 180,E1 -2700.711,E2 -2700.711} C_VEL
LIN {X 0,Y 566.276,Z 553.948,A -85,B 0,C 180,E1 -2702.845,E2 -2702.845} C_VEL
LIN {X 0,Y 566.262,Z 553.952,A -85,B 0,C 180,E1 -2705.698,E2 -2705.698} C_VEL
LIN {X 0,Y 566.231,Z 553.954,A -85,B 0,C 180,E1 -2708.565,E2 -2708.565} C_VEL
LIN {X 0,Y 566.245,Z 553.953,A -85,B 0,C 180,E1 -2711.454,E2 -2711.454} C_VEL
LIN {X 0,Y 566.238,Z 553.953,A -85,B 0,C 180,E1 -2714.506,E2 -2714.506} C_VEL
LIN {X 0,Y 566.202,Z 553.959,A -85,B 0,C 180,E1 -2717.331,E2 -2717.331} C_VEL
LIN {X 0,Y 566.215,Z 553.956,A -85,B 0,C 180,E1 -2720.337,E2 -2720.337} C_VEL
LIN {X 0,Y 566.191,Z 553.961,A -85,B 0,C 180,E1 -2723.403,E2 -2723.403} C_VEL
LIN {X 0,Y 566.217,Z 553.958,A -85,B 0,C 180,E1 -2725.748,E2 -2725.748} C_VEL
LIN {X 0,Y 566.209,Z 553.956,A -85,B 0,C 180,E1 -2727.483,E2 -2727.483} C_VEL
LIN {X 0,Y 565.536,Z 554.044,A -85,B 0,C 180,E1 -2728.077,E2 -2728.077} C_VEL
LIN {X 0,Y 562.669,Z 554.4,A -85,B 0,C 180,E1 -2729.041,E2 -2729.041} C_VEL
LIN {X 0,Y 560.253,Z 554.699,A -85,B 0,C 180,E1 -2729.816,E2 -2729.816} C_VEL
LIN {X 0,Y 559.222,Z 554.83,A -85,B 0,C 180,E1 -2730.415,E2 -2730.415} C_VEL
LIN {X 0,Y 559.141,Z 554.836,A -85,B 0,C 180,E1 -2730.618,E2 -2730.618} C_VEL
LIN {X 0,Y 559.167,Z 554.834,A -85,B 0,C 180,E1 -2733.574,E2 -2733.574} C_VEL
LIN {X 0,Y 559.171,Z 554.835,A -85,B 0,C 180,E1 -2736.448,E2 -2736.448} C_VEL
LIN {X 0,Y 559.179,Z 554.832,A -85,B 0,C 180,E1 -2738.933,E2 -2738.933} C_VEL
LIN {X 0,Y 559.188,Z 554.831,A -85,B 0,C 180,E1 -2741.768,E2 -2741.768} C_VEL
LIN {X 0,Y 559.142,Z 554.838,A -85,B 0,C 180,E1 -2744.739,E2 -2744.739} C_VEL
LIN {X 0,Y 559.165,Z 554.834,A -85,B 0,C 180,E1 -2747.257,E2 -2747.257} C_VEL
LIN {X 0,Y 559.187,Z 554.833,A -85,B 0,C 180,E1 -2750.135,E2 -2750.135} C_VEL
LIN {X 0,Y 559.141,Z 554.837,A -85,B 0,C 180,E1 -2752.891,E2 -2752.891} C_VEL
LIN {X 0,Y 559.166,Z 554.836,A -85,B 0,C 180,E1 -2756.05,E2 -2756.05} C_VEL
LIN {X 0,Y 559.165,Z 554.834,A -85,B 0,C 180,E1 -2758.981,E2 -2758.981} C_VEL
LIN {X 0,Y 559.169,Z 554.834,A -85,B 0,C 180,E1 -2761.618,E2 -2761.618} C_VEL
LIN {X 0,Y 559.183,Z 554.832,A -85,B 0,C 180,E1 -2763.903,E2 -2763.903} C_VEL
LIN {X 0,Y 559.158,Z 554.838,A -85,B 0,C 180,E1 -2766.567,E2 -2766.567} C_VEL
LIN {X 0,Y 559.18,Z 554.831,A -85,B 0,C 180,E1 -2769.395,E2 -2769.395} C_VEL
LIN {X 0,Y 559.148,Z 554.836,A -85,B 0,C 180,E1 -2771.685,E2 -2771.685} C_VEL
LIN {X 0,Y 559.169,Z 554.834,A -85,B 0,C 180,E1 -2773.947,E2 -2773.947} C_VEL
LIN {X 0,Y 559.173,Z 554.834,A -85,B 0,C 180,E1 -2776.184,E2 -2776.184} C_VEL
LIN {X 0,Y 559.196,Z 554.831,A -85,B 0,C 180,E1 -2779.133,E2 -2779.133} C_VEL
LIN {X 0,Y 559.204,Z 554.83,A -85,B 0,C 180,E1 -2782.053,E2 -2782.053} C_VEL
LIN {X 0,Y 559.255,Z 554.824,A -85,B 0,C 180,E1 -2784.953,E2 -2784.953} C_VEL
LIN {X 0,Y 559.255,Z 554.824,A -85,B 0,C 180,E1 -2787.839,E2 -2787.839} C_VEL
LIN {X 0,Y 559.27,Z 554.822,A -85,B 0,C 180,E1 -2790.719,E2 -2790.719} C_VEL
LIN {X 0,Y 559.229,Z 554.827,A -85,B 0,C 180,E1 -2791.845,E2 -2791.845} C_VEL
LIN {X 0,Y 559.758,Z 558.808,A -85,B 0,C 180,E1 -2792.023,E2 -2792.023} C_VEL
LIN {X 0,Y 559.621,Z 569.337,A -85,B 0,C 180,E1 -2792.519,E2 -2792.519} C_VEL
LIN {X 0,Y 559.514,Z 578.593,A -85,B 0,C 180,E1 -2793.059,E2 -2793.059} C_VEL
LIN {X 0,Y 559.377,Z 587.53,A -85,B 0,C 180,E1 -2793.691,E2 -2793.691} C_VEL
LIN {X 0,Y 559.219,Z 595.127,A -85,B 0,C 180,E1 -2794.324,E2 -2794.324} C_VEL
LIN {X 0,Y 559.129,Z 604.096,A -85,B 0,C 180,E1 -2795.228,E2 -2795.228} C_VEL
LIN {X 0,Y 559.058,Z 611.552,A -85,B 0,C 180,E1 -2796.133,E2 -2796.133} C_VEL
LIN {X 0,Y 558.986,Z 617.792,A -85,B 0,C 180,E1 -2797.04,E2 -2797.04} C_VEL
LIN {X 0,Y 558.89,Z 623.014,A -85,B 0,C 180,E1 -2797.95,E2 -2797.95} C_VEL
LIN {X 0,Y 558.838,Z 628.082,A -85,B 0,C 180,E1 -2799.044,E2 -2799.044} C_VEL
LIN {X 0,Y 558.815,Z 632.018,A -85,B 0,C 180,E1 -2800.14,E2 -2800.14} C_VEL
LIN {X 0,Y 558.788,Z 634.789,A -85,B 0,C 180,E1 -2801.182,E2 -2801.182} C_VEL
LIN {X 0,Y 558.768,Z 636.831,A -85,B 0,C 180,E1 -2802.346,E2 -2802.346} C_VEL
LIN {X 0,Y 558.741,Z 637.631,A -85,B 0,C 180,E1 -2803.085,E2 -2803.085} C_VEL
LIN {X 0,Y 558.785,Z 637.886,A -85,B 0,C 180,E1 -2804.432,E2 -2804.432} C_VEL
LIN {X 0,Y 558.714,Z 637.365,A -85,B 0,C 180,E1 -2805.316,E2 -2805.316} C_VEL
LIN {X 0,Y 558.746,Z 636.421,A -85,B 0,C 180,E1 -2806.064,E2 -2806.064} C_VEL
LIN {X 0,Y 558.8,Z 633.176,A -85,B 0,C 180,E1 -2807.568,E2 -2807.568} C_VEL
LIN {X 0,Y 558.812,Z 629.447,A -85,B 0,C 180,E1 -2808.705,E2 -2808.705} C_VEL
LIN {X 0,Y 558.879,Z 624.48,A -85,B 0,C 180,E1 -2809.847,E2 -2809.847} C_VEL
LIN {X 0,Y 558.93,Z 619.285,A -85,B 0,C 180,E1 -2810.806,E2 -2810.806} C_VEL
LIN {X 0,Y 559.013,Z 612.771,A -85,B 0,C 180,E1 -2811.791,E2 -2811.791} C_VEL
LIN {X 0,Y 559.069,Z 606.882,A -85,B 0,C 180,E1 -2812.544,E2 -2812.544} C_VEL
LIN {X 0,Y 559.189,Z 599.289,A -85,B 0,C 180,E1 -2813.366,E2 -2813.366} C_VEL
LIN {X 0,Y 559.289,Z 591.202,A -85,B 0,C 180,E1 -2814.103,E2 -2814.103} C_VEL
LIN {X 0,Y 559.453,Z 582.21,A -85,B 0,C 180,E1 -2814.787,E2 -2814.787} C_VEL
LIN {X 0,Y 559.583,Z 572.854,A -85,B 0,C 180,E1 -2815.377,E2 -2815.377} C_VEL
LIN {X 0,Y 559.661,Z 563.251,A -85,B 0,C 180,E1 -2815.872,E2 -2815.872} C_VEL
LIN {X 0,Y 559.8,Z 557.707,A -85,B 0,C 180,E1 -2816.115,E2 -2816.115} C_VEL
LIN {X 0,Y 559.204,Z 554.83,A -85,B 0,C 180,E1 -2816.245,E2 -2816.245} C_VEL
LIN {X 0,Y 559.16,Z 554.836,A -85,B 0,C 180,E1 -2818.529,E2 -2818.529} C_VEL
LIN {X 0,Y 559.153,Z 554.835,A -85,B 0,C 180,E1 -2821.275,E2 -2821.275} C_VEL
LIN {X 0,Y 559.16,Z 554.837,A -85,B 0,C 180,E1 -2823.949,E2 -2823.949} C_VEL
LIN {X 0,Y 559.139,Z 554.838,A -85,B 0,C 180,E1 -2827.107,E2 -2827.107} C_VEL
LIN {X 0,Y 559.165,Z 554.837,A -85,B 0,C 180,E1 -2829.943,E2 -2829.943} C_VEL
LIN {X 0,Y 559.216,Z 554.905,A -85,B 0,C 180,E1 -2831.328,E2 -2831.328} C_VEL
LIN {X 0,Y 559.327,Z 561.841,A -85,B 0,C 180,E1 -2833.714,E2 -2833.714} C_VEL
LIN {X 0,Y 559.328,Z 569.18,A -85,B 0,C 180,E1 -2836.285,E2 -2836.285} C_VEL
LIN {X 0,Y 559.305,Z 576.685,A -85,B 0,C 180,E1 -2838.931,E2 -2838.931} C_VEL
LIN {X 0,Y 559.23,Z 585.56,A -85,B 0,C 180,E1 -2841.991,E2 -2841.991} C_VEL
LIN {X 0,Y 559.137,Z 593.575,A -85,B 0,C 180,E1 -2844.785,E2 -2844.785} C_VEL
LIN {X 0,Y 559.056,Z 601.1,A -85,B 0,C 180,E1 -2847.379,E2 -2847.379} C_VEL
LIN {X 0,Y 559,Z 609.321,A -85,B 0,C 180,E1 -2850.167,E2 -2850.167} C_VEL
LIN {X 0,Y 558.924,Z 618.055,A -85,B 0,C 180,E1 -2853.085,E2 -2853.085} C_VEL
LIN {X 0,Y 558.938,Z 621.662,A -85,B 0,C 180,E1 -2854.229,E2 -2854.229} C_VEL
LIN {X 0,Y 559.958,Z 629.173,A -85,B 0,C 180,E1 -2854.395,E2 -2854.395} C_VEL
LIN {X 0,Y 559.863,Z 641.164,A -85,B 0,C 180,E1 -2854.735,E2 -2854.735} C_VEL
LIN {X 0,Y 559.72,Z 652.32,A -85,B 0,C 180,E1 -2855.175,E2 -2855.175} C_VEL
LIN {X 0,Y 559.588,Z 662.873,A -85,B 0,C 180,E1 -2855.713,E2 -2855.713} C_VEL
LIN {X 0,Y 559.463,Z 672.163,A -85,B 0,C 180,E1 -2856.298,E2 -2856.298} C_VEL
LIN {X 0,Y 559.324,Z 680.367,A -85,B 0,C 180,E1 -2856.917,E2 -2856.917} C_VEL
LIN {X 0,Y 559.193,Z 688.607,A -85,B 0,C 180,E1 -2857.655,E2 -2857.655} C_VEL
LIN {X 0,Y 559.088,Z 697.535,A -85,B 0,C 180,E1 -2858.621,E2 -2858.621} C_VEL
LIN {X 0,Y 558.947,Z 706.135,A -85,B 0,C 180,E1 -2859.771,E2 -2859.771} C_VEL
LIN {X 0,Y 558.914,Z 712.888,A -85,B 0,C 180,E1 -2860.918,E2 -2860.918} C_VEL
LIN {X 0,Y 558.834,Z 718.152,A -85,B 0,C 180,E1 -2862.055,E2 -2862.055} C_VEL
LIN {X 0,Y 558.809,Z 722.179,A -85,B 0,C 180,E1 -2863.186,E2 -2863.186} C_VEL
LIN {X 0,Y 558.762,Z 724.271,A -85,B 0,C 180,E1 -2863.936,E2 -2863.936} C_VEL
LIN {X 0,Y 558.736,Z 725.851,A -85,B 0,C 180,E1 -2864.684,E2 -2864.684} C_VEL
LIN {X 0,Y 558.766,Z 727.139,A -85,B 0,C 180,E1 -2865.572,E2 -2865.572} C_VEL
LIN {X 0,Y 558.737,Z 727.978,A -85,B 0,C 180,E1 -2866.914,E2 -2866.914} C_VEL
LIN {X 0,Y 558.783,Z 727.284,A -85,B 0,C 180,E1 -2868.391,E2 -2868.391} C_VEL
LIN {X 0,Y 558.827,Z 726.332,A -85,B 0,C 180,E1 -2869.127,E2 -2869.127} C_VEL
LIN {X 0,Y 558.776,Z 723.112,A -85,B 0,C 180,E1 -2870.59,E2 -2870.59} C_VEL
LIN {X 0,Y 558.842,Z 719.527,A -85,B 0,C 180,E1 -2871.685,E2 -2871.685} C_VEL
LIN {X 0,Y 558.882,Z 714.851,A -85,B 0,C 180,E1 -2872.776,E2 -2872.776} C_VEL
LIN {X 0,Y 558.936,Z 708.953,A -85,B 0,C 180,E1 -2873.865,E2 -2873.865} C_VEL
LIN {X 0,Y 559.009,Z 701.65,A -85,B 0,C 180,E1 -2874.951,E2 -2874.951} C_VEL
LIN {X 0,Y 559.115,Z 692.583,A -85,B 0,C 180,E1 -2876.036,E2 -2876.036} C_VEL
LIN {X 0,Y 559.286,Z 683.172,A -85,B 0,C 180,E1 -2876.939,E2 -2876.939} C_VEL
LIN {X 0,Y 559.434,Z 672.767,A -85,B 0,C 180,E1 -2877.75,E2 -2877.75} C_VEL
LIN {X 0,Y 559.537,Z 662.827,A -85,B 0,C 180,E1 -2878.381,E2 -2878.381} C_VEL
LIN {X 0,Y 559.722,Z 652.185,A -85,B 0,C 180,E1 -2878.921,E2 -2878.921} C_VEL
LIN {X 0,Y 559.901,Z 640.679,A -85,B 0,C 180,E1 -2879.371,E2 -2879.371} C_VEL
LIN {X 0,Y 559.818,Z 627.129,A -85,B 0,C 180,E1 -2879.742,E2 -2879.742} C_VEL
LIN {X 0,Y 558.984,Z 621.509,A -85,B 0,C 180,E1 -2879.865,E2 -2879.865} C_VEL
LIN {X 0,Y 559.019,Z 613.545,A -85,B 0,C 180,E1 -2882.522,E2 -2882.522} C_VEL
LIN {X 0,Y 559.07,Z 606.064,A -85,B 0,C 180,E1 -2885.049,E2 -2885.049} C_VEL
LIN {X 0,Y 559.115,Z 597.61,A -85,B 0,C 180,E1 -2887.948,E2 -2887.948} C_VEL
LIN {X 0,Y 559.212,Z 589.256,A -85,B 0,C 180,E1 -2890.866,E2 -2890.866} C_VEL
LIN {X 0,Y 559.271,Z 580.826,A -85,B 0,C 180,E1 -2893.814,E2 -2893.814} C_VEL
LIN {X 0,Y 559.273,Z 574.07,A -85,B 0,C 180,E1 -2896.049,E2 -2896.049} C_VEL
LIN {X 0,Y 559.216,Z 565.733,A -85,B 0,C 180,E1 -2898.692,E2 -2898.692} C_VEL
LIN {X 0,Y 559.076,Z 556.217,A -85,B 0,C 180,E1 -2901.532,E2 -2901.532} C_VEL
LIN {X 0,Y 559.098,Z 554.846,A -85,B 0,C 180,E1 -2901.978,E2 -2901.978} C_VEL
LIN {X 0,Y 559.151,Z 554.838,A -85,B 0,C 180,E1 -2904.506,E2 -2904.506} C_VEL
LIN {X 0,Y 559.175,Z 554.836,A -85,B 0,C 180,E1 -2906.902,E2 -2906.902} C_VEL
LIN {X 0,Y 559.184,Z 554.833,A -85,B 0,C 180,E1 -2909.866,E2 -2909.866} C_VEL
LIN {X 0,Y 559.171,Z 554.834,A -85,B 0,C 180,E1 -2912.715,E2 -2912.715} C_VEL
LIN {X 0,Y 559.155,Z 554.838,A -85,B 0,C 180,E1 -2915.322,E2 -2915.322} C_VEL
LIN {X 0,Y 559.131,Z 554.839,A -85,B 0,C 180,E1 -2918.018,E2 -2918.018} C_VEL
LIN {X 0,Y 559.172,Z 554.835,A -85,B 0,C 180,E1 -2920.811,E2 -2920.811} C_VEL
LIN {X 0,Y 559.159,Z 554.837,A -85,B 0,C 180,E1 -2923.733,E2 -2923.733} C_VEL
LIN {X 0,Y 559.165,Z 554.837,A -85,B 0,C 180,E1 -2926.802,E2 -2926.802} C_VEL
LIN {X 0,Y 559.174,Z 554.835,A -85,B 0,C 180,E1 -2929.19,E2 -2929.19} C_VEL
LIN {X 0,Y 559.134,Z 554.842,A -85,B 0,C 180,E1 -2931.984,E2 -2931.984} C_VEL
LIN {X 0,Y 559.19,Z 554.934,A -85,B 0,C 180,E1 -2932.872,E2 -2932.872} C_VEL
LIN {X 0,Y 560.269,Z 561.261,A -85,B 0,C 180,E1 -2934.294,E2 -2934.294} C_VEL
LIN {X 0,Y 560.229,Z 575.335,A -85,B 0,C 180,E1 -2937.194,E2 -2937.194} C_VEL
LIN {X 0,Y 560.17,Z 589.322,A -85,B 0,C 180,E1 -2939.962,E2 -2939.962} C_VEL
LIN {X 0,Y 560.111,Z 603.716,A -85,B 0,C 180,E1 -2942.709,E2 -2942.709} C_VEL
LIN {X 0,Y 559.978,Z 614.175,A -85,B 0,C 180,E1 -2944.742,E2 -2944.742} C_VEL
LIN {X 0,Y 559.745,Z 627.924,A -85,B 0,C 180,E1 -2947.484,E2 -2947.484} C_VEL
LIN {X 0,Y 559.518,Z 642.83,A -85,B 0,C 180,E1 -2950.401,E2 -2950.401} C_VEL
LIN {X 0,Y 559.322,Z 657.388,A -85,B 0,C 180,E1 -2953.203,E2 -2953.203} C_VEL
LIN {X 0,Y 559.173,Z 673.102,A -85,B 0,C 180,E1 -2956.185,E2 -2956.185} C_VEL
LIN {X 0,Y 559.135,Z 678.141,A -85,B 0,C 180,E1 -2957.132,E2 -2957.132} C_VEL
LIN {X 0,Y 560.032,Z 685.127,A -85,B 0,C 180,E1 -2957.268,E2 -2957.268} C_VEL
LIN {X 0,Y 559.908,Z 698.765,A -85,B 0,C 180,E1 -2957.611,E2 -2957.611} C_VEL
LIN {X 0,Y 559.783,Z 711.54,A -85,B 0,C 180,E1 -2958.091,E2 -2958.091} C_VEL
LIN {X 0,Y 559.59,Z 723.559,A -85,B 0,C 180,E1 -2958.703,E2 -2958.703} C_VEL
LIN {X 0,Y 559.442,Z 734.492,A -85,B 0,C 180,E1 -2959.414,E2 -2959.414} C_VEL
LIN {X 0,Y 559.297,Z 744.655,A -85,B 0,C 180,E1 -2960.234,E2 -2960.234} C_VEL
LIN {X 0,Y 559.134,Z 753.793,A -85,B 0,C 180,E1 -2961.143,E2 -2961.143} C_VEL
LIN {X 0,Y 559.009,Z 762.695,A -85,B 0,C 180,E1 -2962.233,E2 -2962.233} C_VEL
LIN {X 0,Y 558.924,Z 768.746,A -85,B 0,C 180,E1 -2963.14,E2 -2963.14} C_VEL
LIN {X 0,Y 558.935,Z 774.683,A -85,B 0,C 180,E1 -2964.227,E2 -2964.227} C_VEL
LIN {X 0,Y 558.827,Z 779.375,A -85,B 0,C 180,E1 -2965.312,E2 -2965.312} C_VEL
LIN {X 0,Y 558.836,Z 782.959,A -85,B 0,C 180,E1 -2966.396,E2 -2966.396} C_VEL
LIN {X 0,Y 558.799,Z 784.81,A -85,B 0,C 180,E1 -2967.117,E2 -2967.117} C_VEL
LIN {X 0,Y 558.745,Z 787.186,A -85,B 0,C 180,E1 -2968.559,E2 -2968.559} C_VEL
LIN {X 0,Y 558.74,Z 788,A -85,B 0,C 180,E1 -2970.001,E2 -2970.001} C_VEL
LIN {X 0,Y 558.745,Z 787.186,A -85,B 0,C 180,E1 -2971.442,E2 -2971.442} C_VEL
LIN {X 0,Y 558.799,Z 784.808,A -85,B 0,C 180,E1 -2972.884,E2 -2972.884} C_VEL
LIN {X 0,Y 558.844,Z 781.894,A -85,B 0,C 180,E1 -2973.967,E2 -2973.967} C_VEL
LIN {X 0,Y 558.799,Z 777.946,A -85,B 0,C 180,E1 -2975.051,E2 -2975.051} C_VEL
LIN {X 0,Y 558.921,Z 772.864,A -85,B 0,C 180,E1 -2976.136,E2 -2976.136} C_VEL
LIN {X 0,Y 558.978,Z 766.464,A -85,B 0,C 180,E1 -2977.223,E2 -2977.223} C_VEL
LIN {X 0,Y 559.097,Z 758.473,A -85,B 0,C 180,E1 -2978.312,E2 -2978.312} C_VEL
LIN {X 0,Y 559.195,Z 750.33,A -85,B 0,C 180,E1 -2979.222,E2 -2979.222} C_VEL
LIN {X 0,Y 559.352,Z 740.394,A -85,B 0,C 180,E1 -2980.132,E2 -2980.132} C_VEL
LIN {X 0,Y 559.538,Z 729.396,A -85,B 0,C 180,E1 -2980.937,E2 -2980.937} C_VEL
LIN {X 0,Y 559.673,Z 717.452,A -85,B 0,C 180,E1 -2981.628,E2 -2981.628} C_VEL
LIN {X 0,Y 559.814,Z 704.751,A -85,B 0,C 180,E1 -2982.185,E2 -2982.185} C_VEL
LIN {X 0,Y 559.99,Z 691.325,A -85,B 0,C 180,E1 -2982.596,E2 -2982.596} C_VEL
LIN {X 0,Y 559.823,Z 682.573,A -85,B 0,C 180,E1 -2982.784,E2 -2982.784} C_VEL
LIN {X 0,Y 559.113,Z 678.031,A -85,B 0,C 180,E1 -2982.893,E2 -2982.893} C_VEL
LIN {X 0,Y 559.257,Z 663.358,A -85,B 0,C 180,E1 -2985.676,E2 -2985.676} C_VEL
LIN {X 0,Y 559.425,Z 649.663,A -85,B 0,C 180,E1 -2988.305,E2 -2988.305} C_VEL
LIN {X 0,Y 559.636,Z 635.969,A -85,B 0,C 180,E1 -2990.972,E2 -2990.972} C_VEL
LIN {X 0,Y 559.843,Z 622.274,A -85,B 0,C 180,E1 -2993.686,E2 -2993.686} C_VEL
LIN {X 0,Y 560.071,Z 608.428,A -85,B 0,C 180,E1 -2996.454,E2 -2996.454} C_VEL
LIN {X 0,Y 560.149,Z 593.734,A -85,B 0,C 180,E1 -2999.296,E2 -2999.296} C_VEL
LIN {X 0,Y 560.21,Z 579.975,A -85,B 0,C 180,E1 -3002.009,E2 -3002.009} C_VEL
LIN {X 0,Y 560.286,Z 567.373,A -85,B 0,C 180,E1 -3004.583,E2 -3004.583} C_VEL
LIN {X 0,Y 560.18,Z 560.128,A -85,B 0,C 180,E1 -3006.133,E2 -3006.133} C_VEL
LIN {X 0,Y 559.159,Z 554.838,A -85,B 0,C 180,E1 -3007.352,E2 -3007.352} C_VEL
LIN {X 0,Y 559.17,Z 554.836,A -85,B 0,C 180,E1 -3009.942,E2 -3009.942} C_VEL
LIN {X 0,Y 559.166,Z 554.834,A -85,B 0,C 180,E1 -3012.743,E2 -3012.743} C_VEL
LIN {X 0,Y 559.157,Z 554.837,A -85,B 0,C 180,E1 -3015.761,E2 -3015.761} C_VEL
LIN {X 0,Y 559.189,Z 554.832,A -85,B 0,C 180,E1 -3018.232,E2 -3018.232} C_VEL
LIN {X 0,Y 559.177,Z 554.834,A -85,B 0,C 180,E1 -3021.192,E2 -3021.192} C_VEL
LIN {X 0,Y 559.178,Z 554.835,A -85,B 0,C 180,E1 -3023.792,E2 -3023.792} C_VEL
LIN {X 0,Y 559.168,Z 554.835,A -85,B 0,C 180,E1 -3026.425,E2 -3026.425} C_VEL
LIN {X 0,Y 559.159,Z 554.834,A -85,B 0,C 180,E1 -3028.981,E2 -3028.981} C_VEL
LIN {X 0,Y 559.175,Z 554.833,A -85,B 0,C 180,E1 -3031.618,E2 -3031.618} C_VEL
LIN {X 0,Y 559.186,Z 554.832,A -85,B 0,C 180,E1 -3033.903,E2 -3033.903} C_VEL
LIN {X 0,Y 559.146,Z 554.839,A -85,B 0,C 180,E1 -3036.571,E2 -3036.571} C_VEL
LIN {X 0,Y 559.184,Z 554.831,A -85,B 0,C 180,E1 -3039.395,E2 -3039.395} C_VEL
LIN {X 0,Y 559.149,Z 554.836,A -85,B 0,C 180,E1 -3041.686,E2 -3041.686} C_VEL
LIN {X 0,Y 559.172,Z 554.834,A -85,B 0,C 180,E1 -3043.948,E2 -3043.948} C_VEL
LIN {X 0,Y 559.175,Z 554.835,A -85,B 0,C 180,E1 -3046.184,E2 -3046.184} C_VEL
LIN {X 0,Y 559.197,Z 554.831,A -85,B 0,C 180,E1 -3049.133,E2 -3049.133} C_VEL
LIN {X 0,Y 559.209,Z 554.83,A -85,B 0,C 180,E1 -3052.053,E2 -3052.053} C_VEL
LIN {X 0,Y 559.259,Z 554.823,A -85,B 0,C 180,E1 -3054.953,E2 -3054.953} C_VEL
LIN {X 0,Y 559.25,Z 554.826,A -85,B 0,C 180,E1 -3057.839,E2 -3057.839} C_VEL
LIN {X 0,Y 559.277,Z 554.821,A -85,B 0,C 180,E1 -3060.72,E2 -3060.72} C_VEL
LIN {X 0,Y 559.242,Z 554.824,A -85,B 0,C 180,E1 -3062.881,E2 -3062.881} C_VEL
LIN {X 0,Y 559.232,Z 554.828,A -85,B 0,C 180,E1 -3065.77,E2 -3065.77} C_VEL
LIN {X 0,Y 559.19,Z 554.831,A -85,B 0,C 180,E1 -3068.674,E2 -3068.674} C_VEL
LIN {X 0,Y 559.208,Z 554.831,A -85,B 0,C 180,E1 -3071.6,E2 -3071.6} C_VEL
LIN {X 0,Y 559.203,Z 554.83,A -85,B 0,C 180,E1 -3074.595,E2 -3074.595} C_VEL
LIN {X 0,Y 559.161,Z 554.837,A -85,B 0,C 180,E1 -3077.557,E2 -3077.557} C_VEL
LIN {X 0,Y 559.174,Z 554.835,A -85,B 0,C 180,E1 -3079.837,E2 -3079.837} C_VEL
LIN {X 0,Y 559.145,Z 554.839,A -85,B 0,C 180,E1 -3082.152,E2 -3082.152} C_VEL
LIN {X 0,Y 559.182,Z 554.832,A -85,B 0,C 180,E1 -3085.187,E2 -3085.187} C_VEL
LIN {X 0,Y 559.191,Z 554.831,A -85,B 0,C 180,E1 -3087.711,E2 -3087.711} C_VEL
LIN {X 0,Y 559.141,Z 554.836,A -85,B 0,C 180,E1 -3090.618,E2 -3090.618} C_VEL
LIN {X 0,Y 558.48,Z 554.921,A -85,B 0,C 180,E1 -3091.219,E2 -3091.219} C_VEL
LIN {X 0,Y 555.621,Z 555.276,A -85,B 0,C 180,E1 -3092.195,E2 -3092.195} C_VEL
LIN {X 0,Y 553.21,Z 555.576,A -85,B 0,C 180,E1 -3092.981,E2 -3092.981} C_VEL
LIN {X 0,Y 552.191,Z 555.703,A -85,B 0,C 180,E1 -3093.588,E2 -3093.588} C_VEL
LIN {X 0,Y 552.117,Z 555.712,A -85,B 0,C 180,E1 -3093.793,E2 -3093.793} C_VEL
LIN {X 0,Y 552.114,Z 555.713,A -85,B 0,C 180,E1 -3096.746,E2 -3096.746} C_VEL
LIN {X 0,Y 552.133,Z 555.711,A -85,B 0,C 180,E1 -3099.526,E2 -3099.526} C_VEL
LIN {X 0,Y 552.132,Z 555.711,A -85,B 0,C 180,E1 -3102.425,E2 -3102.425} C_VEL
LIN {X 0,Y 552.101,Z 555.716,A -85,B 0,C 180,E1 -3105.562,E2 -3105.562} C_VEL
LIN {X 0,Y 552.142,Z 555.71,A -85,B 0,C 180,E1 -3108.676,E2 -3108.676} C_VEL
LIN {X 0,Y 552.122,Z 555.713,A -85,B 0,C 180,E1 -3111.411,E2 -3111.411} C_VEL
LIN {X 0,Y 552.086,Z 555.716,A -85,B 0,C 180,E1 -3114.156,E2 -3114.156} C_VEL
LIN {X 0,Y 552.122,Z 555.712,A -85,B 0,C 180,E1 -3116.814,E2 -3116.814} C_VEL
LIN {X 0,Y 552.109,Z 555.715,A -85,B 0,C 180,E1 -3119.391,E2 -3119.391} C_VEL
LIN {X 0,Y 552.121,Z 555.714,A -85,B 0,C 180,E1 -3121.902,E2 -3121.902} C_VEL
LIN {X 0,Y 552.157,Z 555.708,A -85,B 0,C 180,E1 -3124.649,E2 -3124.649} C_VEL
LIN {X 0,Y 552.097,Z 555.716,A -85,B 0,C 180,E1 -3127.549,E2 -3127.549} C_VEL
LIN {X 0,Y 552.157,Z 555.707,A -85,B 0,C 180,E1 -3130.674,E2 -3130.674} C_VEL
LIN {X 0,Y 552.119,Z 555.714,A -85,B 0,C 180,E1 -3133.737,E2 -3133.737} C_VEL
LIN {X 0,Y 552.136,Z 555.712,A -85,B 0,C 180,E1 -3136.004,E2 -3136.004} C_VEL
LIN {X 0,Y 552.163,Z 555.707,A -85,B 0,C 180,E1 -3138.993,E2 -3138.993} C_VEL
LIN {X 0,Y 552.158,Z 555.709,A -85,B 0,C 180,E1 -3141.951,E2 -3141.951} C_VEL
LIN {X 0,Y 552.23,Z 555.699,A -85,B 0,C 180,E1 -3144.888,E2 -3144.888} C_VEL
LIN {X 0,Y 552.226,Z 555.7,A -85,B 0,C 180,E1 -3147.811,E2 -3147.811} C_VEL
LIN {X 0,Y 552.24,Z 555.698,A -85,B 0,C 180,E1 -3150.729,E2 -3150.729} C_VEL
LIN {X 0,Y 552.209,Z 555.855,A -85,B 0,C 180,E1 -3151.731,E2 -3151.731} C_VEL
LIN {X 0,Y 552.801,Z 559.723,A -85,B 0,C 180,E1 -3151.912,E2 -3151.912} C_VEL
LIN {X 0,Y 552.641,Z 569.265,A -85,B 0,C 180,E1 -3152.368,E2 -3152.368} C_VEL
LIN {X 0,Y 552.509,Z 578.537,A -85,B 0,C 180,E1 -3152.916,E2 -3152.916} C_VEL
LIN {X 0,Y 552.362,Z 587.481,A -85,B 0,C 180,E1 -3153.555,E2 -3153.555} C_VEL
LIN {X 0,Y 552.189,Z 595.089,A -85,B 0,C 180,E1 -3154.196,E2 -3154.196} C_VEL
LIN {X 0,Y 552.086,Z 604.06,A -85,B 0,C 180,E1 -3155.112,E2 -3155.112} C_VEL
LIN {X 0,Y 551.953,Z 610.201,A -85,B 0,C 180,E1 -3155.846,E2 -3155.846} C_VEL
LIN {X 0,Y 551.908,Z 616.038,A -85,B 0,C 180,E1 -3156.663,E2 -3156.663} C_VEL
LIN {X 0,Y 551.815,Z 622.082,A -85,B 0,C 180,E1 -3157.684,E2 -3157.684} C_VEL
LIN {X 0,Y 551.775,Z 627.33,A -85,B 0,C 180,E1 -3158.791,E2 -3158.791} C_VEL
LIN {X 0,Y 551.739,Z 631.441,A -85,B 0,C 180,E1 -3159.901,E2 -3159.901} C_VEL
LIN {X 0,Y 551.708,Z 634.949,A -85,B 0,C 180,E1 -3161.226,E2 -3161.226} C_VEL
LIN {X 0,Y 551.667,Z 636.055,A -85,B 0,C 180,E1 -3161.76,E2 -3161.76} C_VEL
LIN {X 0,Y 551.654,Z 637.71,A -85,B 0,C 180,E1 -3163.256,E2 -3163.256} C_VEL
LIN {X 0,Y 551.674,Z 637.997,A -85,B 0,C 180,E1 -3164.007,E2 -3164.007} C_VEL
LIN {X 0,Y 551.614,Z 637.133,A -85,B 0,C 180,E1 -3165.518,E2 -3165.518} C_VEL
LIN {X 0,Y 551.658,Z 636.144,A -85,B 0,C 180,E1 -3166.276,E2 -3166.276} C_VEL
LIN {X 0,Y 551.705,Z 634.286,A -85,B 0,C 180,E1 -3167.177,E2 -3167.177} C_VEL
LIN {X 0,Y 551.715,Z 630.203,A -85,B 0,C 180,E1 -3168.569,E2 -3168.569} C_VEL
LIN {X 0,Y 551.804,Z 625.365,A -85,B 0,C 180,E1 -3169.741,E2 -3169.741} C_VEL
LIN {X 0,Y 551.831,Z 620.468,A -85,B 0,C 180,E1 -3170.696,E2 -3170.696} C_VEL
LIN {X 0,Y 551.95,Z 614.37,A -85,B 0,C 180,E1 -3171.669,E2 -3171.669} C_VEL
LIN {X 0,Y 552.043,Z 606.902,A -85,B 0,C 180,E1 -3172.65,E2 -3172.65} C_VEL
LIN {X 0,Y 552.149,Z 599.961,A -85,B 0,C 180,E1 -3173.419,E2 -3173.419} C_VEL
LIN {X 0,Y 552.273,Z 591.224,A -85,B 0,C 180,E1 -3174.229,E2 -3174.229} C_VEL
LIN {X 0,Y 552.454,Z 582.405,A -85,B 0,C 180,E1 -3174.91,E2 -3174.91} C_VEL
LIN {X 0,Y 552.625,Z 572.603,A -85,B 0,C 180,E1 -3175.534,E2 -3175.534} C_VEL
LIN {X 0,Y 552.703,Z 563.304,A -85,B 0,C 180,E1 -3176.019,E2 -3176.019} C_VEL
LIN {X 0,Y 552.648,Z 557.857,A -85,B 0,C 180,E1 -3176.266,E2 -3176.266} C_VEL
LIN {X 0,Y 552.174,Z 555.705,A -85,B 0,C 180,E1 -3176.376,E2 -3176.376} C_VEL
LIN {X 0,Y 552.112,Z 555.714,A -85,B 0,C 180,E1 -3178.927,E2 -3178.927} C_VEL
LIN {X 0,Y 552.13,Z 555.711,A -85,B 0,C 180,E1 -3181.479,E2 -3181.479} C_VEL
LIN {X 0,Y 552.129,Z 555.712,A -85,B 0,C 180,E1 -3184.17,E2 -3184.17} C_VEL
LIN {X 0,Y 552.109,Z 555.713,A -85,B 0,C 180,E1 -3186.746,E2 -3186.746} C_VEL
LIN {X 0,Y 552.13,Z 555.712,A -85,B 0,C 180,E1 -3189.526,E2 -3189.526} C_VEL
LIN {X 0,Y 552.19,Z 555.861,A -85,B 0,C 180,E1 -3191.261,E2 -3191.261} C_VEL
LIN {X 0,Y 552.298,Z 562.313,A -85,B 0,C 180,E1 -3193.505,E2 -3193.505} C_VEL
LIN {X 0,Y 552.326,Z 569.695,A -85,B 0,C 180,E1 -3196.076,E2 -3196.076} C_VEL
LIN {X 0,Y 552.277,Z 576.925,A -85,B 0,C 180,E1 -3198.659,E2 -3198.659} C_VEL
LIN {X 0,Y 552.173,Z 584.781,A -85,B 0,C 180,E1 -3201.416,E2 -3201.416} C_VEL
LIN {X 0,Y 552.127,Z 592.656,A -85,B 0,C 180,E1 -3204.16,E2 -3204.16} C_VEL
LIN {X 0,Y 552.051,Z 600.213,A -85,B 0,C 180,E1 -3206.81,E2 -3206.81} C_VEL
LIN {X 0,Y 551.959,Z 609.41,A -85,B 0,C 180,E1 -3209.976,E2 -3209.976} C_VEL
LIN {X 0,Y 551.857,Z 618.507,A -85,B 0,C 180,E1 -3213.055,E2 -3213.055} C_VEL
LIN {X 0,Y 551.845,Z 621.473,A -85,B 0,C 180,E1 -3214.051,E2 -3214.051} C_VEL
LIN {X 0,Y 553.067,Z 630.306,A -85,B 0,C 180,E1 -3214.264,E2 -3214.264} C_VEL
LIN {X 0,Y 552.922,Z 642.073,A -85,B 0,C 180,E1 -3214.612,E2 -3214.612} C_VEL
LIN {X 0,Y 552.755,Z 652.775,A -85,B 0,C 180,E1 -3215.046,E2 -3215.046} C_VEL
LIN {X 0,Y 552.612,Z 663.176,A -85,B 0,C 180,E1 -3215.586,E2 -3215.586} C_VEL
LIN {X 0,Y 552.44,Z 673.166,A -85,B 0,C 180,E1 -3216.232,E2 -3216.232} C_VEL
LIN {X 0,Y 552.265,Z 683.615,A -85,B 0,C 180,E1 -3217.063,E2 -3217.063} C_VEL
LIN {X 0,Y 552.09,Z 694.374,A -85,B 0,C 180,E1 -3218.14,E2 -3218.14} C_VEL
LIN {X 0,Y 551.942,Z 702.188,A -85,B 0,C 180,E1 -3219.113,E2 -3219.113} C_VEL
LIN {X 0,Y 551.871,Z 707.465,A -85,B 0,C 180,E1 -3219.889,E2 -3219.889} C_VEL
LIN {X 0,Y 551.83,Z 713.917,A -85,B 0,C 180,E1 -3221.049,E2 -3221.049} C_VEL
LIN {X 0,Y 551.737,Z 718.957,A -85,B 0,C 180,E1 -3222.199,E2 -3222.199} C_VEL
LIN {X 0,Y 551.701,Z 722.787,A -85,B 0,C 180,E1 -3223.344,E2 -3223.344} C_VEL
LIN {X 0,Y 551.635,Z 725.51,A -85,B 0,C 180,E1 -3224.482,E2 -3224.482} C_VEL
LIN {X 0,Y 551.675,Z 727.074,A -85,B 0,C 180,E1 -3225.506,E2 -3225.506} C_VEL
LIN {X 0,Y 551.651,Z 727.937,A -85,B 0,C 180,E1 -3226.743,E2 -3226.743} C_VEL
LIN {X 0,Y 551.674,Z 727.464,A -85,B 0,C 180,E1 -3228.239,E2 -3228.239} C_VEL
LIN {X 0,Y 551.733,Z 726.578,A -85,B 0,C 180,E1 -3228.985,E2 -3228.985} C_VEL
LIN {X 0,Y 551.689,Z 723.593,A -85,B 0,C 180,E1 -3230.468,E2 -3230.468} C_VEL
LIN {X 0,Y 551.742,Z 720.17,A -85,B 0,C 180,E1 -3231.577,E2 -3231.577} C_VEL
LIN {X 0,Y 551.8,Z 715.655,A -85,B 0,C 180,E1 -3232.683,E2 -3232.683} C_VEL
LIN {X 0,Y 551.796,Z 710.736,A -85,B 0,C 180,E1 -3233.651,E2 -3233.651} C_VEL
LIN {X 0,Y 551.863,Z 704.141,A -85,B 0,C 180,E1 -3234.703,E2 -3234.703} C_VEL
LIN {X 0,Y 552.021,Z 697.176,A -85,B 0,C 180,E1 -3235.619,E2 -3235.619} C_VEL
LIN {X 0,Y 552.148,Z 688.813,A -85,B 0,C 180,E1 -3236.534,E2 -3236.534} C_VEL
LIN {X 0,Y 552.312,Z 679.727,A -85,B 0,C 180,E1 -3237.356,E2 -3237.356} C_VEL
LIN {X 0,Y 552.498,Z 668.582,A -85,B 0,C 180,E1 -3238.178,E2 -3238.178} C_VEL
LIN {X 0,Y 552.683,Z 657.602,A -85,B 0,C 180,E1 -3238.816,E2 -3238.816} C_VEL
LIN {X 0,Y 552.889,Z 645.205,A -85,B 0,C 180,E1 -3239.363,E2 -3239.363} C_VEL
LIN {X 0,Y 552.991,Z 634.051,A -85,B 0,C 180,E1 -3239.727,E2 -3239.727} C_VEL
LIN {X 0,Y 552.841,Z 627.47,A -85,B 0,C 180,E1 -3239.898,E2 -3239.898} C_VEL
LIN {X 0,Y 551.893,Z 621.47,A -85,B 0,C 180,E1 -3240.046,E2 -3240.046} C_VEL
LIN {X 0,Y 551.961,Z 614.046,A -85,B 0,C 180,E1 -3242.555,E2 -3242.555} C_VEL
LIN {X 0,Y 552.022,Z 606.566,A -85,B 0,C 180,E1 -3245.113,E2 -3245.113} C_VEL
LIN {X 0,Y 552.067,Z 598.115,A -85,B 0,C 180,E1 -3248.05,E2 -3248.05} C_VEL
LIN {X 0,Y 552.161,Z 590.755,A -85,B 0,C 180,E1 -3250.636,E2 -3250.636} C_VEL
LIN {X 0,Y 552.212,Z 583.312,A -85,B 0,C 180,E1 -3253.244,E2 -3253.244} C_VEL
LIN {X 0,Y 552.225,Z 576.584,A -85,B 0,C 180,E1 -3255.502,E2 -3255.502} C_VEL
LIN {X 0,Y 552.188,Z 568.257,A -85,B 0,C 180,E1 -3258.17,E2 -3258.17} C_VEL
LIN {X 0,Y 552.051,Z 560.651,A -85,B 0,C 180,E1 -3260.493,E2 -3260.493} C_VEL
LIN {X 0,Y 552.043,Z 555.725,A -85,B 0,C 180,E1 -3261.961,E2 -3261.961} C_VEL
LIN {X 0,Y 552.102,Z 555.718,A -85,B 0,C 180,E1 -3264.038,E2 -3264.038} C_VEL
LIN {X 0,Y 552.13,Z 555.712,A -85,B 0,C 180,E1 -3266.456,E2 -3266.456} C_VEL
LIN {X 0,Y 552.113,Z 555.715,A -85,B 0,C 180,E1 -3268.928,E2 -3268.928} C_VEL
LIN {X 0,Y 552.13,Z 555.712,A -85,B 0,C 180,E1 -3271.481,E2 -3271.481} C_VEL
LIN {X 0,Y 552.142,Z 555.711,A -85,B 0,C 180,E1 -3274.173,E2 -3274.173} C_VEL
LIN {X 0,Y 552.113,Z 555.713,A -85,B 0,C 180,E1 -3276.747,E2 -3276.747} C_VEL
LIN {X 0,Y 552.13,Z 555.713,A -85,B 0,C 180,E1 -3279.527,E2 -3279.527} C_VEL
LIN {X 0,Y 552.127,Z 555.711,A -85,B 0,C 180,E1 -3282.426,E2 -3282.426} C_VEL
LIN {X 0,Y 552.096,Z 555.717,A -85,B 0,C 180,E1 -3285.564,E2 -3285.564} C_VEL
LIN {X 0,Y 552.137,Z 555.711,A -85,B 0,C 180,E1 -3288.677,E2 -3288.677} C_VEL
LIN {X 0,Y 552.118,Z 555.714,A -85,B 0,C 180,E1 -3291.412,E2 -3291.412} C_VEL
LIN {X 0,Y 552.133,Z 555.756,A -85,B 0,C 180,E1 -3292.628,E2 -3292.628} C_VEL
LIN {X 0,Y 553.371,Z 562.843,A -85,B 0,C 180,E1 -3294.254,E2 -3294.254} C_VEL
LIN {X 0,Y 553.301,Z 575.775,A -85,B 0,C 180,E1 -3296.964,E2 -3296.964} C_VEL
LIN {X 0,Y 553.169,Z 591.024,A -85,B 0,C 180,E1 -3300.028,E2 -3300.028} C_VEL
LIN {X 0,Y 553.084,Z 605.366,A -85,B 0,C 180,E1 -3302.809,E2 -3302.809} C_VEL
LIN {X 0,Y 552.95,Z 620.058,A -85,B 0,C 180,E1 -3305.603,E2 -3305.603} C_VEL
LIN {X 0,Y 552.705,Z 633.817,A -85,B 0,C 180,E1 -3308.362,E2 -3308.362} C_VEL
LIN {X 0,Y 552.431,Z 649.531,A -85,B 0,C 180,E1 -3311.456,E2 -3311.456} C_VEL
LIN {X 0,Y 552.23,Z 665.245,A -85,B 0,C 180,E1 -3314.5,E2 -3314.5} C_VEL
LIN {X 0,Y 552.074,Z 678.141,A -85,B 0,C 180,E1 -3316.965,E2 -3316.965} C_VEL
LIN {X 0,Y 553.121,Z 686.268,A -85,B 0,C 180,E1 -3317.13,E2 -3317.13} C_VEL
LIN {X 0,Y 552.949,Z 699.525,A -85,B 0,C 180,E1 -3317.476,E2 -3317.476} C_VEL
LIN {X 0,Y 552.794,Z 712.524,A -85,B 0,C 180,E1 -3317.985,E2 -3317.985} C_VEL
LIN {X 0,Y 552.608,Z 724.208,A -85,B 0,C 180,E1 -3318.597,E2 -3318.597} C_VEL
LIN {X 0,Y 552.426,Z 735.756,A -85,B 0,C 180,E1 -3319.371,E2 -3319.371} C_VEL
LIN {X 0,Y 552.232,Z 746.609,A -85,B 0,C 180,E1 -3320.293,E2 -3320.293} C_VEL
LIN {X 0,Y 552.079,Z 755.42,A -85,B 0,C 180,E1 -3321.214,E2 -3321.214} C_VEL
LIN {X 0,Y 551.949,Z 764.007,A -85,B 0,C 180,E1 -3322.317,E2 -3322.317} C_VEL
LIN {X 0,Y 551.822,Z 770.872,A -85,B 0,C 180,E1 -3323.419,E2 -3323.419} C_VEL
LIN {X 0,Y 551.804,Z 776.369,A -85,B 0,C 180,E1 -3324.519,E2 -3324.519} C_VEL
LIN {X 0,Y 551.764,Z 780.68,A -85,B 0,C 180,E1 -3325.618,E2 -3325.618} C_VEL
LIN {X 0,Y 551.75,Z 782.96,A -85,B 0,C 180,E1 -3326.349,E2 -3326.349} C_VEL
LIN {X 0,Y 551.724,Z 784.81,A -85,B 0,C 180,E1 -3327.08,E2 -3327.08} C_VEL
LIN {X 0,Y 551.645,Z 787.186,A -85,B 0,C 180,E1 -3328.541,E2 -3328.541} C_VEL
LIN {X 0,Y 551.64,Z 788,A -85,B 0,C 180,E1 -3330.001,E2 -3330.001} C_VEL
LIN {X 0,Y 551.645,Z 787.185,A -85,B 0,C 180,E1 -3331.461,E2 -3331.461} C_VEL
LIN {X 0,Y 551.724,Z 784.808,A -85,B 0,C 180,E1 -3332.921,E2 -3332.921} C_VEL
LIN {X 0,Y 551.764,Z 781.894,A -85,B 0,C 180,E1 -3334.018,E2 -3334.018} C_VEL
LIN {X 0,Y 551.724,Z 777.946,A -85,B 0,C 180,E1 -3335.116,E2 -3335.116} C_VEL
LIN {X 0,Y 551.803,Z 772.191,A -85,B 0,C 180,E1 -3336.341,E2 -3336.341} C_VEL
LIN {X 0,Y 551.927,Z 765.233,A -85,B 0,C 180,E1 -3337.5,E2 -3337.5} C_VEL
LIN {X 0,Y 552.078,Z 756.986,A -85,B 0,C 180,E1 -3338.603,E2 -3338.603} C_VEL
LIN {X 0,Y 552.201,Z 748.533,A -85,B 0,C 180,E1 -3339.524,E2 -3339.524} C_VEL
LIN {X 0,Y 552.412,Z 738.09,A -85,B 0,C 180,E1 -3340.446,E2 -3340.446} C_VEL
LIN {X 0,Y 552.612,Z 727.3,A -85,B 0,C 180,E1 -3341.213,E2 -3341.213} C_VEL
LIN {X 0,Y 552.747,Z 716.398,A -85,B 0,C 180,E1 -3341.831,E2 -3341.831} C_VEL
LIN {X 0,Y 552.896,Z 704.747,A -85,B 0,C 180,E1 -3342.34,E2 -3342.34} C_VEL
LIN {X 0,Y 553.069,Z 691.324,A -85,B 0,C 180,E1 -3342.756,E2 -3342.756} C_VEL
LIN {X 0,Y 552.913,Z 683.46,A -85,B 0,C 180,E1 -3342.932,E2 -3342.932} C_VEL
LIN {X 0,Y 552.059,Z 678.031,A -85,B 0,C 180,E1 -3343.06,E2 -3343.06} C_VEL
LIN {X 0,Y 552.231,Z 663.358,A -85,B 0,C 180,E1 -3345.88,E2 -3345.88} C_VEL
LIN {X 0,Y 552.433,Z 649.663,A -85,B 0,C 180,E1 -3348.545,E2 -3348.545} C_VEL
LIN {X 0,Y 552.65,Z 635.969,A -85,B 0,C 180,E1 -3351.25,E2 -3351.25} C_VEL
LIN {X 0,Y 552.904,Z 622.274,A -85,B 0,C 180,E1 -3354.002,E2 -3354.002} C_VEL
LIN {X 0,Y 553.059,Z 607.889,A -85,B 0,C 180,E1 -3356.8,E2 -3356.8} C_VEL
LIN {X 0,Y 553.171,Z 594.155,A -85,B 0,C 180,E1 -3359.493,E2 -3359.493} C_VEL
LIN {X 0,Y 553.263,Z 582.013,A -85,B 0,C 180,E1 -3361.911,E2 -3361.911} C_VEL
LIN {X 0,Y 553.372,Z 569.208,A -85,B 0,C 180,E1 -3364.559,E2 -3364.559} C_VEL
LIN {X 0,Y 553.25,Z 561.594,A -85,B 0,C 180,E1 -3366.207,E2 -3366.207} C_VEL
LIN {X 0,Y 552.103,Z 555.717,A -85,B 0,C 180,E1 -3367.606,E2 -3367.606} C_VEL
LIN {X 0,Y 552.126,Z 555.712,A -85,B 0,C 180,E1 -3370.48,E2 -3370.48} C_VEL
LIN {X 0,Y 552.124,Z 555.713,A -85,B 0,C 180,E1 -3373.485,E2 -3373.485} C_VEL
LIN {X 0,Y 552.115,Z 555.714,A -85,B 0,C 180,E1 -3376.577,E2 -3376.577} C_VEL
LIN {X 0,Y 552.114,Z 555.713,A -85,B 0,C 180,E1 -3379.519,E2 -3379.519} C_VEL
LIN {X 0,Y 552.096,Z 555.716,A -85,B 0,C 180,E1 -3382.336,E2 -3382.336} C_VEL
LIN {X 0,Y 552.134,Z 555.711,A -85,B 0,C 180,E1 -3385.054,E2 -3385.054} C_VEL
LIN {X 0,Y 552.119,Z 555.712,A -85,B 0,C 180,E1 -3387.681,E2 -3387.681} C_VEL
LIN {X 0,Y 552.116,Z 555.712,A -85,B 0,C 180,E1 -3390.235,E2 -3390.235} C_VEL
LIN {X 0,Y 552.145,Z 555.711,A -85,B 0,C 180,E1 -3392.999,E2 -3392.999} C_VEL
LIN {X 0,Y 552.118,Z 555.713,A -85,B 0,C 180,E1 -3395.161,E2 -3395.161} C_VEL
LIN {X 0,Y 552.13,Z 555.711,A -85,B 0,C 180,E1 -3398.337,E2 -3398.337} C_VEL
LIN {X 0,Y 552.16,Z 555.707,A -85,B 0,C 180,E1 -3400.674,E2 -3400.674} C_VEL
LIN {X 0,Y 552.122,Z 555.714,A -85,B 0,C 180,E1 -3403.737,E2 -3403.737} C_VEL
LIN {X 0,Y 552.139,Z 555.712,A -85,B 0,C 180,E1 -3406.004,E2 -3406.004} C_VEL
LIN {X 0,Y 552.165,Z 555.706,A -85,B 0,C 180,E1 -3408.993,E2 -3408.993} C_VEL
LIN {X 0,Y 552.164,Z 555.709,A -85,B 0,C 180,E1 -3411.951,E2 -3411.951} C_VEL
LIN {X 0,Y 552.234,Z 555.698,A -85,B 0,C 180,E1 -3414.889,E2 -3414.889} C_VEL
LIN {X 0,Y 552.222,Z 555.701,A -85,B 0,C 180,E1 -3417.812,E2 -3417.812} C_VEL
LIN {X 0,Y 552.247,Z 555.696,A -85,B 0,C 180,E1 -3420.729,E2 -3420.729} C_VEL
LIN {X 0,Y 552.208,Z 555.701,A -85,B 0,C 180,E1 -3422.918,E2 -3422.918} C_VEL
LIN {X 0,Y 552.202,Z 555.704,A -85,B 0,C 180,E1 -3425.844,E2 -3425.844} C_VEL
LIN {X 0,Y 552.161,Z 555.707,A -85,B 0,C 180,E1 -3428.785,E2 -3428.785} C_VEL
LIN {X 0,Y 552.166,Z 555.708,A -85,B 0,C 180,E1 -3431.75,E2 -3431.75} C_VEL
LIN {X 0,Y 552.14,Z 555.71,A -85,B 0,C 180,E1 -3434.748,E2 -3434.748} C_VEL
LIN {X 0,Y 552.113,Z 555.714,A -85,B 0,C 180,E1 -3437.788,E2 -3437.788} C_VEL
LIN {X 0,Y 552.133,Z 555.712,A -85,B 0,C 180,E1 -3440.101,E2 -3440.101} C_VEL
LIN {X 0,Y 552.099,Z 555.716,A -85,B 0,C 180,E1 -3442.45,E2 -3442.45} C_VEL
LIN {X 0,Y 552.158,Z 555.707,A -85,B 0,C 180,E1 -3445.35,E2 -3445.35} C_VEL
LIN {X 0,Y 552.125,Z 555.714,A -85,B 0,C 180,E1 -3448.097,E2 -3448.097} C_VEL
LIN {X 0,Y 552.104,Z 555.715,A -85,B 0,C 180,E1 -3450.614,E2 -3450.614} C_VEL
LIN {X 0,Y 552.124,Z 555.711,A -85,B 0,C 180,E1 -3453.185,E2 -3453.185} C_VEL
LIN {X 0,Y 552.117,Z 555.712,A -85,B 0,C 180,E1 -3453.793,E2 -3453.793} C_VEL
LIN {X 0,Y 551.481,Z 555.793,A -85,B 0,C 180,E1 -3454.402,E2 -3454.402} C_VEL
LIN {X 0,Y 548.66,Z 556.145,A -85,B 0,C 180,E1 -3455.39,E2 -3455.39} C_VEL
LIN {X 0,Y 546.239,Z 556.447,A -85,B 0,C 180,E1 -3456.186,E2 -3456.186} C_VEL
LIN {X 0,Y 545.17,Z 556.578,A -85,B 0,C 180,E1 -3456.8,E2 -3456.8} C_VEL
LIN {X 0,Y 545.067,Z 556.591,A -85,B 0,C 180,E1 -3457.007,E2 -3457.007} C_VEL
LIN {X 0,Y 545.073,Z 556.59,A -85,B 0,C 180,E1 -3460.142,E2 -3460.142} C_VEL
LIN {X 0,Y 545.088,Z 556.59,A -85,B 0,C 180,E1 -3463.105,E2 -3463.105} C_VEL
LIN {X 0,Y 545.066,Z 556.591,A -85,B 0,C 180,E1 -3466.224,E2 -3466.224} C_VEL
LIN {X 0,Y 545.099,Z 556.588,A -85,B 0,C 180,E1 -3468.886,E2 -3468.886} C_VEL
LIN {X 0,Y 545.055,Z 556.592,A -85,B 0,C 180,E1 -3471.762,E2 -3471.762} C_VEL
LIN {X 0,Y 545.037,Z 556.595,A -85,B 0,C 180,E1 -3474.531,E2 -3474.531} C_VEL
LIN {X 0,Y 545.082,Z 556.59,A -85,B 0,C 180,E1 -3477.212,E2 -3477.212} C_VEL
LIN {X 0,Y 545.067,Z 556.592,A -85,B 0,C 180,E1 -3479.81,E2 -3479.81} C_VEL
LIN {X 0,Y 545.09,Z 556.588,A -85,B 0,C 180,E1 -3482.344,E2 -3482.344} C_VEL
LIN {X 0,Y 545.118,Z 556.584,A -85,B 0,C 180,E1 -3484.82,E2 -3484.82} C_VEL
LIN {X 0,Y 545.045,Z 556.593,A -85,B 0,C 180,E1 -3487.242,E2 -3487.242} C_VEL
LIN {X 0,Y 545.121,Z 556.585,A -85,B 0,C 180,E1 -3490.414,E2 -3490.414} C_VEL
LIN {X 0,Y 545.075,Z 556.591,A -85,B 0,C 180,E1 -3493.521,E2 -3493.521} C_VEL
LIN {X 0,Y 545.096,Z 556.588,A -85,B 0,C 180,E1 -3495.819,E2 -3495.819} C_VEL
LIN {X 0,Y 545.119,Z 556.584,A -85,B 0,C 180,E1 -3498.849,E2 -3498.849} C_VEL
LIN {X 0,Y 545.128,Z 556.585,A -85,B 0,C 180,E1 -3501.846,E2 -3501.846} C_VEL
LIN {X 0,Y 545.205,Z 556.573,A -85,B 0,C 180,E1 -3504.822,E2 -3504.822} C_VEL
LIN {X 0,Y 545.197,Z 556.576,A -85,B 0,C 180,E1 -3507.783,E2 -3507.783} C_VEL
LIN {X 0,Y 545.211,Z 556.574,A -85,B 0,C 180,E1 -3510.738,E2 -3510.738} C_VEL
LIN {X 0,Y 545.118,Z 556.585,A -85,B 0,C 180,E1 -3511.546,E2 -3511.546} C_VEL
LIN {X 0,Y 545.93,Z 560.512,A -85,B 0,C 180,E1 -3511.751,E2 -3511.751} C_VEL
LIN {X 0,Y 545.737,Z 569.998,A -85,B 0,C 180,E1 -3512.213,E2 -3512.213} C_VEL
LIN {X 0,Y 545.583,Z 579.175,A -85,B 0,C 180,E1 -3512.768,E2 -3512.768} C_VEL
LIN {X 0,Y 545.412,Z 588.006,A -85,B 0,C 180,E1 -3513.416,E2 -3513.416} C_VEL
LIN {X 0,Y 545.232,Z 595.503,A -85,B 0,C 180,E1 -3514.065,E2 -3514.065} C_VEL
LIN {X 0,Y 545.062,Z 604.321,A -85,B 0,C 180,E1 -3514.992,E2 -3514.992} C_VEL
LIN {X 0,Y 544.908,Z 610.351,A -85,B 0,C 180,E1 -3515.736,E2 -3515.736} C_VEL
LIN {X 0,Y 544.836,Z 616.665,A -85,B 0,C 180,E1 -3516.666,E2 -3516.666} C_VEL
LIN {X 0,Y 544.743,Z 622.967,A -85,B 0,C 180,E1 -3517.785,E2 -3517.785} C_VEL
LIN {X 0,Y 544.675,Z 628.038,A -85,B 0,C 180,E1 -3518.907,E2 -3518.907} C_VEL
LIN {X 0,Y 544.643,Z 631.979,A -85,B 0,C 180,E1 -3520.031,E2 -3520.031} C_VEL
LIN {X 0,Y 544.615,Z 635.097,A -85,B 0,C 180,E1 -3521.264,E2 -3521.264} C_VEL
LIN {X 0,Y 544.56,Z 636.334,A -85,B 0,C 180,E1 -3521.916,E2 -3521.916} C_VEL
LIN {X 0,Y 544.565,Z 637.273,A -85,B 0,C 180,E1 -3522.673,E2 -3522.673} C_VEL
LIN {X 0,Y 544.603,Z 637.97,A -85,B 0,C 180,E1 -3524.192,E2 -3524.192} C_VEL
LIN {X 0,Y 544.546,Z 637.653,A -85,B 0,C 180,E1 -3524.958,E2 -3524.958} C_VEL
LIN {X 0,Y 544.58,Z 635.789,A -85,B 0,C 180,E1 -3526.493,E2 -3526.493} C_VEL
LIN {X 0,Y 544.626,Z 633.182,A -85,B 0,C 180,E1 -3527.652,E2 -3527.652} C_VEL
LIN {X 0,Y 544.667,Z 629.46,A -85,B 0,C 180,E1 -3528.818,E2 -3528.818} C_VEL
LIN {X 0,Y 544.738,Z 624.691,A -85,B 0,C 180,E1 -3529.952,E2 -3529.952} C_VEL
LIN {X 0,Y 544.773,Z 619.302,A -85,B 0,C 180,E1 -3530.976,E2 -3530.976} C_VEL
LIN {X 0,Y 544.904,Z 613.078,A -85,B 0,C 180,E1 -3531.964,E2 -3531.964} C_VEL
LIN {X 0,Y 545.012,Z 607.171,A -85,B 0,C 180,E1 -3532.758,E2 -3532.758} C_VEL
LIN {X 0,Y 545.154,Z 600.192,A -85,B 0,C 180,E1 -3533.555,E2 -3533.555} C_VEL
LIN {X 0,Y 545.301,Z 591.816,A -85,B 0,C 180,E1 -3534.356,E2 -3534.356} C_VEL
LIN {X 0,Y 545.522,Z 582.985,A -85,B 0,C 180,E1 -3535.057,E2 -3535.057} C_VEL
LIN {X 0,Y 545.707,Z 574.076,A -85,B 0,C 180,E1 -3535.644,E2 -3535.644} C_VEL
LIN {X 0,Y 545.83,Z 564.351,A -85,B 0,C 180,E1 -3536.166,E2 -3536.166} C_VEL
LIN {X 0,Y 545.82,Z 559.417,A -85,B 0,C 180,E1 -3536.395,E2 -3536.395} C_VEL
LIN {X 0,Y 545.138,Z 556.582,A -85,B 0,C 180,E1 -3536.544,E2 -3536.544} C_VEL
LIN {X 0,Y 545.078,Z 556.592,A -85,B 0,C 180,E1 -3539.337,E2 -3539.337} C_VEL
LIN {X 0,Y 545.068,Z 556.591,A -85,B 0,C 180,E1 -3541.913,E2 -3541.913} C_VEL
LIN {X 0,Y 545.071,Z 556.59,A -85,B 0,C 180,E1 -3544.563,E2 -3544.563} C_VEL
LIN {X 0,Y 545.035,Z 556.596,A -85,B 0,C 180,E1 -3547.303,E2 -3547.303} C_VEL
LIN {X 0,Y 545.089,Z 556.59,A -85,B 0,C 180,E1 -3550.139,E2 -3550.139} C_VEL
LIN {X 0,Y 545.123,Z 556.592,A -85,B 0,C 180,E1 -3551.109,E2 -3551.109} C_VEL
LIN {X 0,Y 545.307,Z 562.203,A -85,B 0,C 180,E1 -3553.083,E2 -3553.083} C_VEL
LIN {X 0,Y 545.307,Z 570.2,A -85,B 0,C 180,E1 -3555.897,E2 -3555.897} C_VEL
LIN {X 0,Y 545.265,Z 577.246,A -85,B 0,C 180,E1 -3558.379,E2 -3558.379} C_VEL
LIN {X 0,Y 545.149,Z 584.103,A -85,B 0,C 180,E1 -3560.825,E2 -3560.825} C_VEL
LIN {X 0,Y 545.099,Z 592.114,A -85,B 0,C 180,E1 -3563.624,E2 -3563.624} C_VEL
LIN {X 0,Y 545.025,Z 599.612,A -85,B 0,C 180,E1 -3566.326,E2 -3566.326} C_VEL
LIN {X 0,Y 544.908,Z 608.33,A -85,B 0,C 180,E1 -3569.373,E2 -3569.373} C_VEL
LIN {X 0,Y 544.838,Z 616.924,A -85,B 0,C 180,E1 -3572.331,E2 -3572.331} C_VEL
LIN {X 0,Y 544.766,Z 621.474,A -85,B 0,C 180,E1 -3573.879,E2 -3573.879} C_VEL
LIN {X 0,Y 546.14,Z 630.522,A -85,B 0,C 180,E1 -3574.105,E2 -3574.105} C_VEL
LIN {X 0,Y 545.985,Z 642.045,A -85,B 0,C 180,E1 -3574.451,E2 -3574.451} C_VEL
LIN {X 0,Y 545.803,Z 653.078,A -85,B 0,C 180,E1 -3574.906,E2 -3574.906} C_VEL
LIN {X 0,Y 545.63,Z 663.475,A -85,B 0,C 180,E1 -3575.456,E2 -3575.456} C_VEL
LIN {X 0,Y 545.444,Z 672.894,A -85,B 0,C 180,E1 -3576.072,E2 -3576.072} C_VEL
LIN {X 0,Y 545.253,Z 682.665,A -85,B 0,C 180,E1 -3576.851,E2 -3576.851} C_VEL
LIN {X 0,Y 545.078,Z 692.798,A -85,B 0,C 180,E1 -3577.844,E2 -3577.844} C_VEL
LIN {X 0,Y 544.943,Z 700.913,A -85,B 0,C 180,E1 -3578.832,E2 -3578.832} C_VEL
LIN {X 0,Y 544.793,Z 707.688,A -85,B 0,C 180,E1 -3579.833,E2 -3579.833} C_VEL
LIN {X 0,Y 544.767,Z 713.058,A -85,B 0,C 180,E1 -3580.794,E2 -3580.794} C_VEL
LIN {X 0,Y 544.68,Z 718.281,A -85,B 0,C 180,E1 -3581.961,E2 -3581.961} C_VEL
LIN {X 0,Y 544.631,Z 722.273,A -85,B 0,C 180,E1 -3583.122,E2 -3583.122} C_VEL
LIN {X 0,Y 544.56,Z 725.148,A -85,B 0,C 180,E1 -3584.275,E2 -3584.275} C_VEL
LIN {X 0,Y 544.574,Z 727.013,A -85,B 0,C 180,E1 -3585.442,E2 -3585.442} C_VEL
LIN {X 0,Y 544.549,Z 727.861,A -85,B 0,C 180,E1 -3586.567,E2 -3586.567} C_VEL
LIN {X 0,Y 544.561,Z 727.941,A -85,B 0,C 180,E1 -3587.327,E2 -3587.327} C_VEL
LIN {X 0,Y 544.563,Z 727.6,A -85,B 0,C 180,E1 -3588.083,E2 -3588.083} C_VEL
LIN {X 0,Y 544.653,Z 726.779,A -85,B 0,C 180,E1 -3588.84,E2 -3588.84} C_VEL
LIN {X 0,Y 544.602,Z 725.606,A -85,B 0,C 180,E1 -3589.592,E2 -3589.592} C_VEL
LIN {X 0,Y 544.606,Z 723.005,A -85,B 0,C 180,E1 -3590.717,E2 -3590.717} C_VEL
LIN {X 0,Y 544.688,Z 719.383,A -85,B 0,C 180,E1 -3591.841,E2 -3591.841} C_VEL
LIN {X 0,Y 544.719,Z 714.675,A -85,B 0,C 180,E1 -3592.96,E2 -3592.96} C_VEL
LIN {X 0,Y 544.827,Z 708.736,A -85,B 0,C 180,E1 -3594.077,E2 -3594.077} C_VEL
LIN {X 0,Y 544.867,Z 702.705,A -85,B 0,C 180,E1 -3595.005,E2 -3595.005} C_VEL
LIN {X 0,Y 544.987,Z 695.485,A -85,B 0,C 180,E1 -3595.933,E2 -3595.933} C_VEL
LIN {X 0,Y 545.177,Z 686.805,A -85,B 0,C 180,E1 -3596.86,E2 -3596.86} C_VEL
LIN {X 0,Y 545.396,Z 676.117,A -85,B 0,C 180,E1 -3597.785,E2 -3597.785} C_VEL
LIN {X 0,Y 545.553,Z 665.357,A -85,B 0,C 180,E1 -3598.524,E2 -3598.524} C_VEL
LIN {X 0,Y 545.749,Z 655.324,A -85,B 0,C 180,E1 -3599.078,E2 -3599.078} C_VEL
LIN {X 0,Y 545.958,Z 644.721,A -85,B 0,C 180,E1 -3599.539,E2 -3599.539} C_VEL
LIN {X 0,Y 546.086,Z 633.376,A -85,B 0,C 180,E1 -3599.908,E2 -3599.908} C_VEL
LIN {X 0,Y 545.919,Z 628.302,A -85,B 0,C 180,E1 -3600.046,E2 -3600.046} C_VEL
LIN {X 0,Y 544.827,Z 621.497,A -85,B 0,C 180,E1 -3600.208,E2 -3600.208} C_VEL
LIN {X 0,Y 544.877,Z 614.55,A -85,B 0,C 180,E1 -3602.588,E2 -3602.588} C_VEL
LIN {X 0,Y 544.976,Z 607.068,A -85,B 0,C 180,E1 -3605.18,E2 -3605.18} C_VEL
LIN {X 0,Y 545.036,Z 598.631,A -85,B 0,C 180,E1 -3608.155,E2 -3608.155} C_VEL
LIN {X 0,Y 545.106,Z 592.32,A -85,B 0,C 180,E1 -3610.399,E2 -3610.399} C_VEL
LIN {X 0,Y 545.177,Z 584.74,A -85,B 0,C 180,E1 -3613.038,E2 -3613.038} C_VEL
LIN {X 0,Y 545.173,Z 576.84,A -85,B 0,C 180,E1 -3615.707,E2 -3615.707} C_VEL
LIN {X 0,Y 545.127,Z 568.403,A -85,B 0,C 180,E1 -3618.413,E2 -3618.413} C_VEL
LIN {X 0,Y 545.014,Z 558.182,A -85,B 0,C 180,E1 -3621.488,E2 -3621.488} C_VEL
LIN {X 0,Y 545.013,Z 556.601,A -85,B 0,C 180,E1 -3621.96,E2 -3621.96} C_VEL
LIN {X 0,Y 545.047,Z 556.595,A -85,B 0,C 180,E1 -3624.37,E2 -3624.37} C_VEL
LIN {X 0,Y 545.097,Z 556.589,A -85,B 0,C 180,E1 -3627.176,E2 -3627.176} C_VEL
LIN {X 0,Y 545.091,Z 556.59,A -85,B 0,C 180,E1 -3630.251,E2 -3630.251} C_VEL
LIN {X 0,Y 545.088,Z 556.589,A -85,B 0,C 180,E1 -3633.065,E2 -3633.065} C_VEL
LIN {X 0,Y 545.059,Z 556.592,A -85,B 0,C 180,E1 -3635.678,E2 -3635.678} C_VEL
LIN {X 0,Y 545.05,Z 556.594,A -85,B 0,C 180,E1 -3638.238,E2 -3638.238} C_VEL
LIN {X 0,Y 545.097,Z 556.587,A -85,B 0,C 180,E1 -3641.114,E2 -3641.114} C_VEL
LIN {X 0,Y 545.055,Z 556.592,A -85,B 0,C 180,E1 -3644.13,E2 -3644.13} C_VEL
LIN {X 0,Y 545.083,Z 556.591,A -85,B 0,C 180,E1 -3646.895,E2 -3646.895} C_VEL
LIN {X 0,Y 545.09,Z 556.591,A -85,B 0,C 180,E1 -3649.861,E2 -3649.861} C_VEL
LIN {X 0,Y 545.072,Z 556.73,A -85,B 0,C 180,E1 -3652.409,E2 -3652.409} C_VEL
LIN {X 0,Y 546.424,Z 564.049,A -85,B 0,C 180,E1 -3654.125,E2 -3654.125} C_VEL
LIN {X 0,Y 546.356,Z 576.233,A -85,B 0,C 180,E1 -3656.733,E2 -3656.733} C_VEL
LIN {X 0,Y 546.178,Z 591.628,A -85,B 0,C 180,E1 -3659.88,E2 -3659.88} C_VEL
LIN {X 0,Y 546.055,Z 605.574,A -85,B 0,C 180,E1 -3662.632,E2 -3662.632} C_VEL
LIN {X 0,Y 545.921,Z 620.32,A -85,B 0,C 180,E1 -3665.471,E2 -3665.471} C_VEL
LIN {X 0,Y 545.774,Z 631.855,A -85,B 0,C 180,E1 -3667.675,E2 -3667.675} C_VEL
LIN {X 0,Y 545.54,Z 645.603,A -85,B 0,C 180,E1 -3670.431,E2 -3670.431} C_VEL
LIN {X 0,Y 545.25,Z 661.317,A -85,B 0,C 180,E1 -3673.528,E2 -3673.528} C_VEL
LIN {X 0,Y 545.025,Z 677.031,A -85,B 0,C 180,E1 -3676.58,E2 -3676.58} C_VEL
LIN {X 0,Y 545.024,Z 678.139,A -85,B 0,C 180,E1 -3676.793,E2 -3676.793} C_VEL
LIN {X 0,Y 546.19,Z 686.267,A -85,B 0,C 180,E1 -3676.964,E2 -3676.964} C_VEL
LIN {X 0,Y 546.034,Z 699.526,A -85,B 0,C 180,E1 -3677.315,E2 -3677.315} C_VEL
LIN {X 0,Y 545.886,Z 711.53,A -85,B 0,C 180,E1 -3677.783,E2 -3677.783} C_VEL
LIN {X 0,Y 545.654,Z 723.023,A -85,B 0,C 180,E1 -3678.379,E2 -3678.379} C_VEL
LIN {X 0,Y 545.481,Z 734.495,A -85,B 0,C 180,E1 -3679.14,E2 -3679.14} C_VEL
LIN {X 0,Y 545.275,Z 744.655,A -85,B 0,C 180,E1 -3679.98,E2 -3679.98} C_VEL
LIN {X 0,Y 545.081,Z 753.793,A -85,B 0,C 180,E1 -3680.913,E2 -3680.913} C_VEL
LIN {X 0,Y 544.916,Z 762.694,A -85,B 0,C 180,E1 -3682.031,E2 -3682.031} C_VEL
LIN {X 0,Y 544.784,Z 769.853,A -85,B 0,C 180,E1 -3683.147,E2 -3683.147} C_VEL
LIN {X 0,Y 544.741,Z 776.369,A -85,B 0,C 180,E1 -3684.448,E2 -3684.448} C_VEL
LIN {X 0,Y 544.66,Z 780.68,A -85,B 0,C 180,E1 -3685.56,E2 -3685.56} C_VEL
LIN {X 0,Y 544.669,Z 782.96,A -85,B 0,C 180,E1 -3686.302,E2 -3686.302} C_VEL
LIN {X 0,Y 544.65,Z 784.809,A -85,B 0,C 180,E1 -3687.042,E2 -3687.042} C_VEL
LIN {X 0,Y 544.546,Z 787.185,A -85,B 0,C 180,E1 -3688.522,E2 -3688.522} C_VEL
LIN {X 0,Y 544.541,Z 788,A -85,B 0,C 180,E1 -3690.001,E2 -3690.001} C_VEL
LIN {X 0,Y 544.546,Z 787.185,A -85,B 0,C 180,E1 -3691.48,E2 -3691.48} C_VEL
LIN {X 0,Y 544.651,Z 784.808,A -85,B 0,C 180,E1 -3692.959,E2 -3692.959} C_VEL
LIN {X 0,Y 544.684,Z 781.894,A -85,B 0,C 180,E1 -3694.07,E2 -3694.07} C_VEL
LIN {X 0,Y 544.654,Z 777.946,A -85,B 0,C 180,E1 -3695.183,E2 -3695.183} C_VEL
LIN {X 0,Y 544.74,Z 772.705,A -85,B 0,C 180,E1 -3696.328,E2 -3696.328} C_VEL
LIN {X 0,Y 544.837,Z 766.464,A -85,B 0,C 180,E1 -3697.412,E2 -3697.412} C_VEL
LIN {X 0,Y 545.004,Z 758.473,A -85,B 0,C 180,E1 -3698.529,E2 -3698.529} C_VEL
LIN {X 0,Y 545.142,Z 750.329,A -85,B 0,C 180,E1 -3699.461,E2 -3699.461} C_VEL
LIN {X 0,Y 545.363,Z 740.393,A -85,B 0,C 180,E1 -3700.395,E2 -3700.395} C_VEL
LIN {X 0,Y 545.574,Z 730.58,A -85,B 0,C 180,E1 -3701.142,E2 -3701.142} C_VEL
LIN {X 0,Y 545.695,Z 719.579,A -85,B 0,C 180,E1 -3701.817,E2 -3701.817} C_VEL
LIN {X 0,Y 545.909,Z 707.092,A -85,B 0,C 180,E1 -3702.406,E2 -3702.406} C_VEL
LIN {X 0,Y 546.118,Z 694.066,A -85,B 0,C 180,E1 -3702.85,E2 -3702.85} C_VEL
LIN {X 0,Y 546.004,Z 684.345,A -85,B 0,C 180,E1 -3703.081,E2 -3703.081} C_VEL
LIN {X 0,Y 545.023,Z 678.031,A -85,B 0,C 180,E1 -3703.232,E2 -3703.232} C_VEL
LIN {X 0,Y 545.234,Z 663.358,A -85,B 0,C 180,E1 -3706.09,E2 -3706.09} C_VEL
LIN {X 0,Y 545.428,Z 649.663,A -85,B 0,C 180,E1 -3708.792,E2 -3708.792} C_VEL
LIN {X 0,Y 545.677,Z 635.969,A -85,B 0,C 180,E1 -3711.535,E2 -3711.535} C_VEL
LIN {X 0,Y 545.867,Z 624.842,A -85,B 0,C 180,E1 -3713.723,E2 -3713.723} C_VEL
LIN {X 0,Y 546.066,Z 610.17,A -85,B 0,C 180,E1 -3716.567,E2 -3716.567} C_VEL
LIN {X 0,Y 546.172,Z 595.473,A -85,B 0,C 180,E1 -3719.485,E2 -3719.485} C_VEL
LIN {X 0,Y 546.296,Z 583.606,A -85,B 0,C 180,E1 -3721.888,E2 -3721.888} C_VEL
LIN {X 0,Y 546.457,Z 570.742,A -85,B 0,C 180,E1 -3724.603,E2 -3724.603} C_VEL
LIN {X 0,Y 546.331,Z 563.051,A -85,B 0,C 180,E1 -3726.281,E2 -3726.281} C_VEL
LIN {X 0,Y 545.079,Z 556.591,A -85,B 0,C 180,E1 -3727.825,E2 -3727.825} C_VEL
LIN {X 0,Y 545.096,Z 556.588,A -85,B 0,C 180,E1 -3730.474,E2 -3730.474} C_VEL
LIN {X 0,Y 545.083,Z 556.59,A -85,B 0,C 180,E1 -3733.107,E2 -3733.107} C_VEL
LIN {X 0,Y 545.062,Z 556.591,A -85,B 0,C 180,E1 -3736.225,E2 -3736.225} C_VEL
LIN {X 0,Y 545.091,Z 556.589,A -85,B 0,C 180,E1 -3738.886,E2 -3738.886} C_VEL
LIN {X 0,Y 545.055,Z 556.593,A -85,B 0,C 180,E1 -3741.763,E2 -3741.763} C_VEL
LIN {X 0,Y 545.07,Z 556.59,A -85,B 0,C 180,E1 -3744.534,E2 -3744.534} C_VEL
LIN {X 0,Y 545.073,Z 556.591,A -85,B 0,C 180,E1 -3747.212,E2 -3747.212} C_VEL
LIN {X 0,Y 545.068,Z 556.592,A -85,B 0,C 180,E1 -3749.81,E2 -3749.81} C_VEL
LIN {X 0,Y 545.098,Z 556.587,A -85,B 0,C 180,E1 -3752.344,E2 -3752.344} C_VEL
LIN {X 0,Y 545.122,Z 556.583,A -85,B 0,C 180,E1 -3754.82,E2 -3754.82} C_VEL
LIN {X 0,Y 545.042,Z 556.592,A -85,B 0,C 180,E1 -3757.242,E2 -3757.242} C_VEL
LIN {X 0,Y 545.125,Z 556.584,A -85,B 0,C 180,E1 -3760.415,E2 -3760.415} C_VEL
LIN {X 0,Y 545.078,Z 556.59,A -85,B 0,C 180,E1 -3763.521,E2 -3763.521} C_VEL
LIN {X 0,Y 545.099,Z 556.587,A -85,B 0,C 180,E1 -3765.82,E2 -3765.82} C_VEL
LIN {X 0,Y 545.121,Z 556.583,A -85,B 0,C 180,E1 -3768.849,E2 -3768.849} C_VEL
LIN {X 0,Y 545.134,Z 556.584,A -85,B 0,C 180,E1 -3771.847,E2 -3771.847} C_VEL
LIN {X 0,Y 545.21,Z 556.573,A -85,B 0,C 180,E1 -3774.823,E2 -3774.823} C_VEL
LIN {X 0,Y 545.195,Z 556.577,A -85,B 0,C 180,E1 -3777.783,E2 -3777.783} C_VEL
LIN {X 0,Y 545.217,Z 556.572,A -85,B 0,C 180,E1 -3780.738,E2 -3780.738} C_VEL
LIN {X 0,Y 545.175,Z 556.577,A -85,B 0,C 180,E1 -3782.955,E2 -3782.955} C_VEL
LIN {X 0,Y 545.175,Z 556.58,A -85,B 0,C 180,E1 -3785.919,E2 -3785.919} C_VEL
LIN {X 0,Y 545.12,Z 556.584,A -85,B 0,C 180,E1 -3788.9,E2 -3788.9} C_VEL
LIN {X 0,Y 545.138,Z 556.583,A -85,B 0,C 180,E1 -3791.904,E2 -3791.904} C_VEL
LIN {X 0,Y 545.089,Z 556.589,A -85,B 0,C 180,E1 -3794.943,E2 -3794.943} C_VEL
LIN {X 0,Y 545.081,Z 556.589,A -85,B 0,C 180,E1 -3798.025,E2 -3798.025} C_VEL
LIN {X 0,Y 545.098,Z 556.587,A -85,B 0,C 180,E1 -3800.372,E2 -3800.372} C_VEL
LIN {X 0,Y 545.094,Z 556.588,A -85,B 0,C 180,E1 -3803.558,E2 -3803.558} C_VEL
LIN {X 0,Y 545.082,Z 556.589,A -85,B 0,C 180,E1 -3806,E2 -3806} C_VEL
LIN {X 0,Y 545.091,Z 556.588,A -85,B 0,C 180,E1 -3808.748,E2 -3808.748} C_VEL
LIN {X 0,Y 545.061,Z 556.593,A -85,B 0,C 180,E1 -3811.679,E2 -3811.679} C_VEL
LIN {X 0,Y 545.083,Z 556.589,A -85,B 0,C 180,E1 -3814.563,E2 -3814.563} C_VEL
LIN {X 0,Y 545.067,Z 556.591,A -85,B 0,C 180,E1 -3817.007,E2 -3817.007} C_VEL
LIN {X 0,Y 544.359,Z 556.68,A -85,B 0,C 180,E1 -3817.624,E2 -3817.624} C_VEL
LIN {X 0,Y 541.494,Z 557.038,A -85,B 0,C 180,E1 -3818.625,E2 -3818.625} C_VEL
LIN {X 0,Y 539.107,Z 557.333,A -85,B 0,C 180,E1 -3819.431,E2 -3819.431} C_VEL
LIN {X 0,Y 538.098,Z 557.459,A -85,B 0,C 180,E1 -3820.053,E2 -3820.053} C_VEL
LIN {X 0,Y 538.022,Z 557.468,A -85,B 0,C 180,E1 -3820.263,E2 -3820.263} C_VEL
LIN {X 0,Y 538.034,Z 557.468,A -85,B 0,C 180,E1 -3822.988,E2 -3822.988} C_VEL
LIN {X 0,Y 538.03,Z 557.467,A -85,B 0,C 180,E1 -3825.925,E2 -3825.925} C_VEL
LIN {X 0,Y 538.053,Z 557.465,A -85,B 0,C 180,E1 -3829.224,E2 -3829.224} C_VEL
LIN {X 0,Y 537.995,Z 557.471,A -85,B 0,C 180,E1 -3832.122,E2 -3832.122} C_VEL
LIN {X 0,Y 537.999,Z 557.473,A -85,B 0,C 180,E1 -3834.915,E2 -3834.915} C_VEL
LIN {X 0,Y 538.032,Z 557.466,A -85,B 0,C 180,E1 -3837.618,E2 -3837.618} C_VEL
LIN {X 0,Y 538.019,Z 557.468,A -85,B 0,C 180,E1 -3840.238,E2 -3840.238} C_VEL
LIN {X 0,Y 538.064,Z 557.464,A -85,B 0,C 180,E1 -3842.796,E2 -3842.796} C_VEL
LIN {X 0,Y 538.05,Z 557.466,A -85,B 0,C 180,E1 -3845.292,E2 -3845.292} C_VEL
LIN {X 0,Y 538.016,Z 557.47,A -85,B 0,C 180,E1 -3848.041,E2 -3848.041} C_VEL
LIN {X 0,Y 538.038,Z 557.467,A -85,B 0,C 180,E1 -3850.94,E2 -3850.94} C_VEL
LIN {X 0,Y 538.026,Z 557.468,A -85,B 0,C 180,E1 -3853.298,E2 -3853.298} C_VEL
LIN {X 0,Y 538.064,Z 557.463,A -85,B 0,C 180,E1 -3855.63,E2 -3855.63} C_VEL
LIN {X 0,Y 538.078,Z 557.461,A -85,B 0,C 180,E1 -3858.701,E2 -3858.701} C_VEL
LIN {X 0,Y 538.085,Z 557.461,A -85,B 0,C 180,E1 -3861.739,E2 -3861.739} C_VEL
LIN {X 0,Y 538.163,Z 557.451,A -85,B 0,C 180,E1 -3864.754,E2 -3864.754} C_VEL
LIN {X 0,Y 538.169,Z 557.452,A -85,B 0,C 180,E1 -3867.754,E2 -3867.754} C_VEL
LIN {X 0,Y 538.181,Z 557.449,A -85,B 0,C 180,E1 -3870.748,E2 -3870.748} C_VEL
LIN {X 0,Y 538.076,Z 557.463,A -85,B 0,C 180,E1 -3871.379,E2 -3871.379} C_VEL
LIN {X 0,Y 539.044,Z 562.418,A -85,B 0,C 180,E1 -3871.634,E2 -3871.634} C_VEL
LIN {X 0,Y 538.865,Z 572.503,A -85,B 0,C 180,E1 -3872.148,E2 -3872.148} C_VEL
LIN {X 0,Y 538.677,Z 581.418,A -85,B 0,C 180,E1 -3872.71,E2 -3872.71} C_VEL
LIN {X 0,Y 538.481,Z 590.046,A -85,B 0,C 180,E1 -3873.366,E2 -3873.366} C_VEL
LIN {X 0,Y 538.273,Z 598.296,A -85,B 0,C 180,E1 -3874.117,E2 -3874.117} C_VEL
LIN {X 0,Y 538.124,Z 605.282,A -85,B 0,C 180,E1 -3874.869,E2 -3874.869} C_VEL
LIN {X 0,Y 537.974,Z 612.604,A -85,B 0,C 180,E1 -3875.81,E2 -3875.81} C_VEL
LIN {X 0,Y 537.877,Z 618.82,A -85,B 0,C 180,E1 -3876.772,E2 -3876.772} C_VEL
LIN {X 0,Y 537.787,Z 622.934,A -85,B 0,C 180,E1 -3877.508,E2 -3877.508} C_VEL
LIN {X 0,Y 537.672,Z 628.065,A -85,B 0,C 180,E1 -3878.645,E2 -3878.645} C_VEL
LIN {X 0,Y 537.59,Z 632.076,A -85,B 0,C 180,E1 -3879.784,E2 -3879.784} C_VEL
LIN {X 0,Y 537.568,Z 634.229,A -85,B 0,C 180,E1 -3880.546,E2 -3880.546} C_VEL
LIN {X 0,Y 537.492,Z 637.088,A -85,B 0,C 180,E1 -3882.075,E2 -3882.075} C_VEL
LIN {X 0,Y 537.491,Z 637.984,A -85,B 0,C 180,E1 -3882.842,E2 -3882.842} C_VEL
LIN {X 0,Y 537.53,Z 638.373,A -85,B 0,C 180,E1 -3884.383,E2 -3884.383} C_VEL
LIN {X 0,Y 537.485,Z 638.057,A -85,B 0,C 180,E1 -3885.159,E2 -3885.159} C_VEL
LIN {X 0,Y 537.517,Z 635.959,A -85,B 0,C 180,E1 -3886.716,E2 -3886.716} C_VEL
LIN {X 0,Y 537.567,Z 633.265,A -85,B 0,C 180,E1 -3887.892,E2 -3887.892} C_VEL
LIN {X 0,Y 537.624,Z 629.475,A -85,B 0,C 180,E1 -3889.074,E2 -3889.074} C_VEL
LIN {X 0,Y 537.712,Z 626.321,A -85,B 0,C 180,E1 -3889.865,E2 -3889.865} C_VEL
LIN {X 0,Y 537.786,Z 621.483,A -85,B 0,C 180,E1 -3890.861,E2 -3890.861} C_VEL
LIN {X 0,Y 537.935,Z 615.005,A -85,B 0,C 180,E1 -3891.937,E2 -3891.937} C_VEL
LIN {X 0,Y 538.088,Z 608.261,A -85,B 0,C 180,E1 -3892.864,E2 -3892.864} C_VEL
LIN {X 0,Y 538.232,Z 601.294,A -85,B 0,C 180,E1 -3893.672,E2 -3893.672} C_VEL
LIN {X 0,Y 538.4,Z 593.173,A -85,B 0,C 180,E1 -3894.463,E2 -3894.463} C_VEL
LIN {X 0,Y 538.641,Z 584.122,A -85,B 0,C 180,E1 -3895.193,E2 -3895.193} C_VEL
LIN {X 0,Y 538.862,Z 574.093,A -85,B 0,C 180,E1 -3895.853,E2 -3895.853} C_VEL
LIN {X 0,Y 538.971,Z 564.431,A -85,B 0,C 180,E1 -3896.369,E2 -3896.369} C_VEL
LIN {X 0,Y 538.823,Z 560.282,A -85,B 0,C 180,E1 -3896.568,E2 -3896.568} C_VEL
LIN {X 0,Y 538.095,Z 557.461,A -85,B 0,C 180,E1 -3896.716,E2 -3896.716} C_VEL
LIN {X 0,Y 538.038,Z 557.467,A -85,B 0,C 180,E1 -3899.759,E2 -3899.759} C_VEL
LIN {X 0,Y 538.027,Z 557.468,A -85,B 0,C 180,E1 -3902.381,E2 -3902.381} C_VEL
LIN {X 0,Y 538.006,Z 557.472,A -85,B 0,C 180,E1 -3905.083,E2 -3905.083} C_VEL
LIN {X 0,Y 537.989,Z 557.473,A -85,B 0,C 180,E1 -3907.877,E2 -3907.877} C_VEL
LIN {X 0,Y 538.109,Z 557.46,A -85,B 0,C 180,E1 -3910.954,E2 -3910.954} C_VEL
LIN {X 0,Y 538.303,Z 562.395,A -85,B 0,C 180,E1 -3912.757,E2 -3912.757} C_VEL
LIN {X 0,Y 538.28,Z 570.296,A -85,B 0,C 180,E1 -3915.566,E2 -3915.566} C_VEL
LIN {X 0,Y 538.234,Z 577.865,A -85,B 0,C 180,E1 -3918.246,E2 -3918.246} C_VEL
LIN {X 0,Y 538.133,Z 585.015,A -85,B 0,C 180,E1 -3920.787,E2 -3920.787} C_VEL
LIN {X 0,Y 538.074,Z 592.784,A -85,B 0,C 180,E1 -3923.538,E2 -3923.538} C_VEL
LIN {X 0,Y 538.007,Z 600.405,A -85,B 0,C 180,E1 -3926.277,E2 -3926.277} C_VEL
LIN {X 0,Y 537.843,Z 608.981,A -85,B 0,C 180,E1 -3929.362,E2 -3929.362} C_VEL
LIN {X 0,Y 537.755,Z 617.575,A -85,B 0,C 180,E1 -3932.358,E2 -3932.358} C_VEL
LIN {X 0,Y 537.714,Z 621.472,A -85,B 0,C 180,E1 -3933.703,E2 -3933.703} C_VEL
LIN {X 0,Y 539.218,Z 631.482,A -85,B 0,C 180,E1 -3933.963,E2 -3933.963} C_VEL
LIN {X 0,Y 539.057,Z 642.313,A -85,B 0,C 180,E1 -3934.297,E2 -3934.297} C_VEL
LIN {X 0,Y 538.859,Z 652.401,A -85,B 0,C 180,E1 -3934.714,E2 -3934.714} C_VEL
LIN {X 0,Y 538.664,Z 662.069,A -85,B 0,C 180,E1 -3935.22,E2 -3935.22} C_VEL
LIN {X 0,Y 538.478,Z 671.815,A -85,B 0,C 180,E1 -3935.851,E2 -3935.851} C_VEL
LIN {X 0,Y 538.305,Z 680.54,A -85,B 0,C 180,E1 -3936.535,E2 -3936.535} C_VEL
LIN {X 0,Y 538.111,Z 689.114,A -85,B 0,C 180,E1 -3937.339,E2 -3937.339} C_VEL
LIN {X 0,Y 537.953,Z 696.274,A -85,B 0,C 180,E1 -3938.137,E2 -3938.137} C_VEL
LIN {X 0,Y 537.846,Z 702.426,A -85,B 0,C 180,E1 -3938.941,E2 -3938.941} C_VEL
LIN {X 0,Y 537.704,Z 708.817,A -85,B 0,C 180,E1 -3939.935,E2 -3939.935} C_VEL
LIN {X 0,Y 537.671,Z 714.076,A -85,B 0,C 180,E1 -3940.927,E2 -3940.927} C_VEL
LIN {X 0,Y 537.589,Z 719.086,A -85,B 0,C 180,E1 -3942.109,E2 -3942.109} C_VEL
LIN {X 0,Y 537.521,Z 722.881,A -85,B 0,C 180,E1 -3943.283,E2 -3943.283} C_VEL
LIN {X 0,Y 537.466,Z 724.784,A -85,B 0,C 180,E1 -3944.062,E2 -3944.062} C_VEL
LIN {X 0,Y 537.45,Z 726.275,A -85,B 0,C 180,E1 -3944.839,E2 -3944.839} C_VEL
LIN {X 0,Y 537.497,Z 727.242,A -85,B 0,C 180,E1 -3945.616,E2 -3945.616} C_VEL
LIN {X 0,Y 537.467,Z 727.983,A -85,B 0,C 180,E1 -3947.156,E2 -3947.156} C_VEL
LIN {X 0,Y 537.466,Z 727.697,A -85,B 0,C 180,E1 -3947.924,E2 -3947.924} C_VEL
LIN {X 0,Y 537.566,Z 726.981,A -85,B 0,C 180,E1 -3948.691,E2 -3948.691} C_VEL
LIN {X 0,Y 537.516,Z 725.935,A -85,B 0,C 180,E1 -3949.453,E2 -3949.453} C_VEL
LIN {X 0,Y 537.529,Z 723.487,A -85,B 0,C 180,E1 -3950.594,E2 -3950.594} C_VEL
LIN {X 0,Y 537.607,Z 720.025,A -85,B 0,C 180,E1 -3951.733,E2 -3951.733} C_VEL
LIN {X 0,Y 537.634,Z 715.479,A -85,B 0,C 180,E1 -3952.867,E2 -3952.867} C_VEL
LIN {X 0,Y 537.724,Z 709.719,A -85,B 0,C 180,E1 -3953.999,E2 -3953.999} C_VEL
LIN {X 0,Y 537.751,Z 703.887,A -85,B 0,C 180,E1 -3954.939,E2 -3954.939} C_VEL
LIN {X 0,Y 537.926,Z 696.88,A -85,B 0,C 180,E1 -3955.88,E2 -3955.88} C_VEL
LIN {X 0,Y 538.119,Z 688.458,A -85,B 0,C 180,E1 -3956.818,E2 -3956.818} C_VEL
LIN {X 0,Y 538.277,Z 680.398,A -85,B 0,C 180,E1 -3957.568,E2 -3957.568} C_VEL
LIN {X 0,Y 538.471,Z 670.738,A -85,B 0,C 180,E1 -3958.317,E2 -3958.317} C_VEL
LIN {X 0,Y 538.748,Z 658.704,A -85,B 0,C 180,E1 -3959.066,E2 -3959.066} C_VEL
LIN {X 0,Y 539.008,Z 646.714,A -85,B 0,C 180,E1 -3959.627,E2 -3959.627} C_VEL
LIN {X 0,Y 539.159,Z 635.241,A -85,B 0,C 180,E1 -3960.024,E2 -3960.024} C_VEL
LIN {X 0,Y 539.019,Z 629.46,A -85,B 0,C 180,E1 -3960.187,E2 -3960.187} C_VEL
LIN {X 0,Y 537.782,Z 621.523,A -85,B 0,C 180,E1 -3960.375,E2 -3960.375} C_VEL
LIN {X 0,Y 537.832,Z 612.907,A -85,B 0,C 180,E1 -3963.371,E2 -3963.371} C_VEL
LIN {X 0,Y 537.889,Z 606.513,A -85,B 0,C 180,E1 -3965.624,E2 -3965.624} C_VEL
LIN {X 0,Y 538.038,Z 598.302,A -85,B 0,C 180,E1 -3968.64,E2 -3968.64} C_VEL
LIN {X 0,Y 538.106,Z 589.731,A -85,B 0,C 180,E1 -3971.614,E2 -3971.614} C_VEL
LIN {X 0,Y 538.151,Z 581.769,A -85,B 0,C 180,E1 -3974.367,E2 -3974.367} C_VEL
LIN {X 0,Y 538.169,Z 572.252,A -85,B 0,C 180,E1 -3977.479,E2 -3977.479} C_VEL
LIN {X 0,Y 537.995,Z 563.317,A -85,B 0,C 180,E1 -3980.254,E2 -3980.254} C_VEL
LIN {X 0,Y 537.985,Z 557.476,A -85,B 0,C 180,E1 -3982.008,E2 -3982.008} C_VEL
LIN {X 0,Y 538.044,Z 557.468,A -85,B 0,C 180,E1 -3984.708,E2 -3984.708} C_VEL
LIN {X 0,Y 538.06,Z 557.465,A -85,B 0,C 180,E1 -3987.355,E2 -3987.355} C_VEL
LIN {X 0,Y 538.038,Z 557.467,A -85,B 0,C 180,E1 -3989.76,E2 -3989.76} C_VEL
LIN {X 0,Y 538.027,Z 557.469,A -85,B 0,C 180,E1 -3992.382,E2 -3992.382} C_VEL
LIN {X 0,Y 538.017,Z 557.47,A -85,B 0,C 180,E1 -3995.083,E2 -3995.083} C_VEL
LIN {X 0,Y 537.998,Z 557.472,A -85,B 0,C 180,E1 -3997.878,E2 -3997.878} C_VEL
LIN {X 0,Y 538.074,Z 557.463,A -85,B 0,C 180,E1 -4000.774,E2 -4000.774} C_VEL
LIN {X 0,Y 538.025,Z 557.468,A -85,B 0,C 180,E1 -4004.075,E2 -4004.075} C_VEL
LIN {X 0,Y 538.021,Z 557.47,A -85,B 0,C 180,E1 -4007.216,E2 -4007.216} C_VEL
LIN {X 0,Y 538.052,Z 557.466,A -85,B 0,C 180,E1 -4010.207,E2 -4010.207} C_VEL
LIN {X 0,Y 538.029,Z 557.642,A -85,B 0,C 180,E1 -4012.17,E2 -4012.17} C_VEL
LIN {X 0,Y 539.546,Z 565.799,A -85,B 0,C 180,E1 -4014.116,E2 -4014.116} C_VEL
LIN {X 0,Y 539.384,Z 578.226,A -85,B 0,C 180,E1 -4016.823,E2 -4016.823} C_VEL
LIN {X 0,Y 539.202,Z 592.973,A -85,B 0,C 180,E1 -4019.881,E2 -4019.881} C_VEL
LIN {X 0,Y 539.045,Z 606.792,A -85,B 0,C 180,E1 -4022.647,E2 -4022.647} C_VEL
LIN {X 0,Y 538.895,Z 620.547,A -85,B 0,C 180,E1 -4025.335,E2 -4025.335} C_VEL
LIN {X 0,Y 538.707,Z 635.668,A -85,B 0,C 180,E1 -4028.218,E2 -4028.218} C_VEL
LIN {X 0,Y 538.519,Z 647.567,A -85,B 0,C 180,E1 -4030.563,E2 -4030.563} C_VEL
LIN {X 0,Y 538.231,Z 661.317,A -85,B 0,C 180,E1 -4033.306,E2 -4033.306} C_VEL
LIN {X 0,Y 538.032,Z 675.067,A -85,B 0,C 180,E1 -4036.017,E2 -4036.017} C_VEL
LIN {X 0,Y 537.976,Z 678.137,A -85,B 0,C 180,E1 -4036.617,E2 -4036.617} C_VEL
LIN {X 0,Y 539.305,Z 687.407,A -85,B 0,C 180,E1 -4036.818,E2 -4036.818} C_VEL
LIN {X 0,Y 539.105,Z 699.526,A -85,B 0,C 180,E1 -4037.149,E2 -4037.149} C_VEL
LIN {X 0,Y 538.901,Z 712.522,A -85,B 0,C 180,E1 -4037.67,E2 -4037.67} C_VEL
LIN {X 0,Y 538.665,Z 723.966,A -85,B 0,C 180,E1 -4038.283,E2 -4038.283} C_VEL
LIN {X 0,Y 538.502,Z 734.496,A -85,B 0,C 180,E1 -4038.997,E2 -4038.997} C_VEL
LIN {X 0,Y 538.27,Z 744.655,A -85,B 0,C 180,E1 -4039.849,E2 -4039.849} C_VEL
LIN {X 0,Y 538.054,Z 753.793,A -85,B 0,C 180,E1 -4040.793,E2 -4040.793} C_VEL
LIN {X 0,Y 537.85,Z 762.694,A -85,B 0,C 180,E1 -4041.926,E2 -4041.926} C_VEL
LIN {X 0,Y 537.728,Z 769.853,A -85,B 0,C 180,E1 -4043.057,E2 -4043.057} C_VEL
LIN {X 0,Y 537.676,Z 776.369,A -85,B 0,C 180,E1 -4044.375,E2 -4044.375} C_VEL
LIN {X 0,Y 537.557,Z 780.679,A -85,B 0,C 180,E1 -4045.502,E2 -4045.502} C_VEL
LIN {X 0,Y 537.591,Z 782.96,A -85,B 0,C 180,E1 -4046.253,E2 -4046.253} C_VEL
LIN {X 0,Y 537.551,Z 784.809,A -85,B 0,C 180,E1 -4047.003,E2 -4047.003} C_VEL
LIN {X 0,Y 537.451,Z 787.185,A -85,B 0,C 180,E1 -4048.502,E2 -4048.502} C_VEL
LIN {X 0,Y 537.442,Z 788,A -85,B 0,C 180,E1 -4050.001,E2 -4050.001} C_VEL
LIN {X 0,Y 537.451,Z 787.184,A -85,B 0,C 180,E1 -4051.499,E2 -4051.499} C_VEL
LIN {X 0,Y 537.489,Z 786.197,A -85,B 0,C 180,E1 -4052.249,E2 -4052.249} C_VEL
LIN {X 0,Y 537.551,Z 784.809,A -85,B 0,C 180,E1 -4052.998,E2 -4052.998} C_VEL
LIN {X 0,Y 537.603,Z 781.894,A -85,B 0,C 180,E1 -4054.124,E2 -4054.124} C_VEL
LIN {X 0,Y 537.588,Z 777.946,A -85,B 0,C 180,E1 -4055.251,E2 -4055.251} C_VEL
LIN {X 0,Y 537.65,Z 773.081,A -85,B 0,C 180,E1 -4056.335,E2 -4056.335} C_VEL
LIN {X 0,Y 537.792,Z 766.463,A -85,B 0,C 180,E1 -4057.51,E2 -4057.51} C_VEL
LIN {X 0,Y 537.97,Z 758.473,A -85,B 0,C 180,E1 -4058.641,E2 -4058.641} C_VEL
LIN {X 0,Y 538.119,Z 750.328,A -85,B 0,C 180,E1 -4059.586,E2 -4059.586} C_VEL
LIN {X 0,Y 538.353,Z 740.392,A -85,B 0,C 180,E1 -4060.531,E2 -4060.531} C_VEL
LIN {X 0,Y 538.611,Z 730.581,A -85,B 0,C 180,E1 -4061.288,E2 -4061.288} C_VEL
LIN {X 0,Y 538.755,Z 719.505,A -85,B 0,C 180,E1 -4061.975,E2 -4061.975} C_VEL
LIN {X 0,Y 538.988,Z 707.091,A -85,B 0,C 180,E1 -4062.568,E2 -4062.568} C_VEL
LIN {X 0,Y 539.185,Z 694.065,A -85,B 0,C 180,E1 -4063.018,E2 -4063.018} C_VEL
LIN {X 0,Y 539.159,Z 685.628,A -85,B 0,C 180,E1 -4063.223,E2 -4063.223} C_VEL
LIN {X 0,Y 537.971,Z 678.031,A -85,B 0,C 180,E1 -4063.409,E2 -4063.409} C_VEL
LIN {X 0,Y 538.218,Z 663.358,A -85,B 0,C 180,E1 -4066.305,E2 -4066.305} C_VEL
LIN {X 0,Y 538.439,Z 649.663,A -85,B 0,C 180,E1 -4069.046,E2 -4069.046} C_VEL
LIN {X 0,Y 538.653,Z 637.746,A -85,B 0,C 180,E1 -4071.428,E2 -4071.428} C_VEL
LIN {X 0,Y 538.861,Z 622.545,A -85,B 0,C 180,E1 -4074.33,E2 -4074.33} C_VEL
LIN {X 0,Y 539.046,Z 609.393,A -85,B 0,C 180,E1 -4076.941,E2 -4076.941} C_VEL
LIN {X 0,Y 539.189,Z 595.736,A -85,B 0,C 180,E1 -4079.691,E2 -4079.691} C_VEL
LIN {X 0,Y 539.378,Z 582.149,A -85,B 0,C 180,E1 -4082.513,E2 -4082.513} C_VEL
LIN {X 0,Y 539.567,Z 567.608,A -85,B 0,C 180,E1 -4085.654,E2 -4085.654} C_VEL
LIN {X 0,Y 539.047,Z 562.367,A -85,B 0,C 180,E1 -4086.852,E2 -4086.852} C_VEL
LIN {X 0,Y 538.03,Z 557.469,A -85,B 0,C 180,E1 -4088.068,E2 -4088.068} C_VEL
LIN {X 0,Y 538.057,Z 557.466,A -85,B 0,C 180,E1 -4090.776,E2 -4090.776} C_VEL
LIN {X 0,Y 538.035,Z 557.467,A -85,B 0,C 180,E1 -4094.075,E2 -4094.075} C_VEL
LIN {X 0,Y 538.025,Z 557.468,A -85,B 0,C 180,E1 -4097.214,E2 -4097.214} C_VEL
LIN {X 0,Y 538.027,Z 557.47,A -85,B 0,C 180,E1 -4100.203,E2 -4100.203} C_VEL
LIN {X 0,Y 538.034,Z 557.465,A -85,B 0,C 180,E1 -4103.067,E2 -4103.067} C_VEL
LIN {X 0,Y 538.031,Z 557.467,A -85,B 0,C 180,E1 -4105.827,E2 -4105.827} C_VEL
LIN {X 0,Y 538.013,Z 557.471,A -85,B 0,C 180,E1 -4108.499,E2 -4108.499} C_VEL
LIN {X 0,Y 538.065,Z 557.462,A -85,B 0,C 180,E1 -4111.1,E2 -4111.1} C_VEL
LIN {X 0,Y 538.047,Z 557.464,A -85,B 0,C 180,E1 -4113.633,E2 -4113.633} C_VEL
LIN {X 0,Y 538.011,Z 557.469,A -85,B 0,C 180,E1 -4116.122,E2 -4116.122} C_VEL
LIN {X 0,Y 538.044,Z 557.465,A -85,B 0,C 180,E1 -4119.349,E2 -4119.349} C_VEL
LIN {X 0,Y 538.059,Z 557.466,A -85,B 0,C 180,E1 -4122.517,E2 -4122.517} C_VEL
LIN {X 0,Y 538.068,Z 557.461,A -85,B 0,C 180,E1 -4125.63,E2 -4125.63} C_VEL
LIN {X 0,Y 538.081,Z 557.461,A -85,B 0,C 180,E1 -4128.701,E2 -4128.701} C_VEL
LIN {X 0,Y 538.091,Z 557.46,A -85,B 0,C 180,E1 -4131.739,E2 -4131.739} C_VEL
LIN {X 0,Y 538.167,Z 557.45,A -85,B 0,C 180,E1 -4134.755,E2 -4134.755} C_VEL
LIN {X 0,Y 538.167,Z 557.452,A -85,B 0,C 180,E1 -4137.754,E2 -4137.754} C_VEL
LIN {X 0,Y 538.187,Z 557.448,A -85,B 0,C 180,E1 -4140.748,E2 -4140.748} C_VEL
LIN {X 0,Y 538.141,Z 557.453,A -85,B 0,C 180,E1 -4142.994,E2 -4142.994} C_VEL
LIN {X 0,Y 538.128,Z 557.457,A -85,B 0,C 180,E1 -4145.997,E2 -4145.997} C_VEL
LIN {X 0,Y 538.071,Z 557.463,A -85,B 0,C 180,E1 -4149.017,E2 -4149.017} C_VEL
LIN {X 0,Y 538.087,Z 557.461,A -85,B 0,C 180,E1 -4152.062,E2 -4152.062} C_VEL
LIN {X 0,Y 538.049,Z 557.466,A -85,B 0,C 180,E1 -4155.143,E2 -4155.143} C_VEL
LIN {X 0,Y 538.034,Z 557.467,A -85,B 0,C 180,E1 -4158.27,E2 -4158.27} C_VEL
LIN {X 0,Y 538.042,Z 557.466,A -85,B 0,C 180,E1 -4160.651,E2 -4160.651} C_VEL
LIN {X 0,Y 538.027,Z 557.467,A -85,B 0,C 180,E1 -4163.887,E2 -4163.887} C_VEL
LIN {X 0,Y 538.045,Z 557.465,A -85,B 0,C 180,E1 -4166.366,E2 -4166.366} C_VEL
LIN {X 0,Y 538.033,Z 557.468,A -85,B 0,C 180,E1 -4168.933,E2 -4168.933} C_VEL
LIN {X 0,Y 538.015,Z 557.469,A -85,B 0,C 180,E1 -4171.887,E2 -4171.887} C_VEL
LIN {X 0,Y 538.033,Z 557.467,A -85,B 0,C 180,E1 -4174.62,E2 -4174.62} C_VEL
LIN {X 0,Y 538.01,Z 557.471,A -85,B 0,C 180,E1 -4177.17,E2 -4177.17} C_VEL
LIN {X 0,Y 538.022,Z 557.468,A -85,B 0,C 180,E1 -4180.263,E2 -4180.263} C_VEL
LIN {X 0,Y 537.373,Z 557.551,A -85,B 0,C 180,E1 -4180.888,E2 -4180.888} C_VEL
LIN {X 0,Y 534.524,Z 557.906,A -85,B 0,C 180,E1 -4181.903,E2 -4181.903} C_VEL
LIN {X 0,Y 532.101,Z 558.208,A -85,B 0,C 180,E1 -4182.72,E2 -4182.72} C_VEL
LIN {X 0,Y 531.053,Z 558.337,A -85,B 0,C 180,E1 -4183.351,E2 -4183.351} C_VEL
LIN {X 0,Y 530.965,Z 558.347,A -85,B 0,C 180,E1 -4183.565,E2 -4183.565} C_VEL
LIN {X 0,Y 530.968,Z 558.348,A -85,B 0,C 180,E1 -4186.505,E2 -4186.505} C_VEL
LIN {X 0,Y 530.991,Z 558.346,A -85,B 0,C 180,E1 -4188.975,E2 -4188.975} C_VEL
LIN {X 0,Y 530.961,Z 558.349,A -85,B 0,C 180,E1 -4191.529,E2 -4191.529} C_VEL
LIN {X 0,Y 530.955,Z 558.349,A -85,B 0,C 180,E1 -4194.379,E2 -4194.379} C_VEL
LIN {X 0,Y 530.972,Z 558.348,A -85,B 0,C 180,E1 -4197.133,E2 -4197.133} C_VEL
LIN {X 0,Y 530.971,Z 558.348,A -85,B 0,C 180,E1 -4199.803,E2 -4199.803} C_VEL
LIN {X 0,Y 531.016,Z 558.341,A -85,B 0,C 180,E1 -4202.466,E2 -4202.466} C_VEL
LIN {X 0,Y 531.007,Z 558.342,A -85,B 0,C 180,E1 -4204.942,E2 -4204.942} C_VEL
LIN {X 0,Y 530.972,Z 558.346,A -85,B 0,C 180,E1 -4208.246,E2 -4208.246} C_VEL
LIN {X 0,Y 530.996,Z 558.343,A -85,B 0,C 180,E1 -4210.677,E2 -4210.677} C_VEL
LIN {X 0,Y 530.987,Z 558.344,A -85,B 0,C 180,E1 -4213.07,E2 -4213.07} C_VEL
LIN {X 0,Y 531.019,Z 558.339,A -85,B 0,C 180,E1 -4215.435,E2 -4215.435} C_VEL
LIN {X 0,Y 531.049,Z 558.337,A -85,B 0,C 180,E1 -4218.549,E2 -4218.549} C_VEL
LIN {X 0,Y 531.055,Z 558.337,A -85,B 0,C 180,E1 -4221.629,E2 -4221.629} C_VEL
LIN {X 0,Y 531.122,Z 558.328,A -85,B 0,C 180,E1 -4224.685,E2 -4224.685} C_VEL
LIN {X 0,Y 531.141,Z 558.327,A -85,B 0,C 180,E1 -4227.724,E2 -4227.724} C_VEL
LIN {X 0,Y 531.151,Z 558.325,A -85,B 0,C 180,E1 -4230.757,E2 -4230.757} C_VEL
LIN {X 0,Y 531.053,Z 558.339,A -85,B 0,C 180,E1 -4231.208,E2 -4231.208} C_VEL
LIN {X 0,Y 532.106,Z 562.37,A -85,B 0,C 180,E1 -4231.418,E2 -4231.418} C_VEL
LIN {X 0,Y 532.006,Z 573.409,A -85,B 0,C 180,E1 -4231.987,E2 -4231.987} C_VEL
LIN {X 0,Y 531.777,Z 583.659,A -85,B 0,C 180,E1 -4232.651,E2 -4232.651} C_VEL
LIN {X 0,Y 531.496,Z 593.199,A -85,B 0,C 180,E1 -4233.411,E2 -4233.411} C_VEL
LIN {X 0,Y 531.301,Z 602.914,A -85,B 0,C 180,E1 -4234.361,E2 -4234.361} C_VEL
LIN {X 0,Y 531.025,Z 612.267,A -85,B 0,C 180,E1 -4235.505,E2 -4235.505} C_VEL
LIN {X 0,Y 530.922,Z 619.06,A -85,B 0,C 180,E1 -4236.54,E2 -4236.54} C_VEL
LIN {X 0,Y 530.791,Z 624.8,A -85,B 0,C 180,E1 -4237.608,E2 -4237.608} C_VEL
LIN {X 0,Y 530.65,Z 629.765,A -85,B 0,C 180,E1 -4238.76,E2 -4238.76} C_VEL
LIN {X 0,Y 530.575,Z 633.614,A -85,B 0,C 180,E1 -4239.915,E2 -4239.915} C_VEL
LIN {X 0,Y 530.567,Z 635.667,A -85,B 0,C 180,E1 -4240.686,E2 -4240.686} C_VEL
LIN {X 0,Y 530.534,Z 637.205,A -85,B 0,C 180,E1 -4241.46,E2 -4241.46} C_VEL
LIN {X 0,Y 530.471,Z 639.121,A -85,B 0,C 180,E1 -4243.015,E2 -4243.015} C_VEL
LIN {X 0,Y 530.484,Z 639.434,A -85,B 0,C 180,E1 -4243.795,E2 -4243.795} C_VEL
LIN {X 0,Y 530.476,Z 638.898,A -85,B 0,C 180,E1 -4245.364,E2 -4245.364} C_VEL
LIN {X 0,Y 530.496,Z 637.985,A -85,B 0,C 180,E1 -4246.152,E2 -4246.152} C_VEL
LIN {X 0,Y 530.57,Z 634.865,A -85,B 0,C 180,E1 -4247.737,E2 -4247.737} C_VEL
LIN {X 0,Y 530.642,Z 631.264,A -85,B 0,C 180,E1 -4248.934,E2 -4248.934} C_VEL
LIN {X 0,Y 530.749,Z 626.449,A -85,B 0,C 180,E1 -4250.137,E2 -4250.137} C_VEL
LIN {X 0,Y 530.853,Z 621.407,A -85,B 0,C 180,E1 -4251.146,E2 -4251.146} C_VEL
LIN {X 0,Y 530.994,Z 615.594,A -85,B 0,C 180,E1 -4252.107,E2 -4252.107} C_VEL
LIN {X 0,Y 531.162,Z 609.351,A -85,B 0,C 180,E1 -4252.974,E2 -4252.974} C_VEL
LIN {X 0,Y 531.358,Z 601.328,A -85,B 0,C 180,E1 -4253.902,E2 -4253.902} C_VEL
LIN {X 0,Y 531.533,Z 592.864,A -85,B 0,C 180,E1 -4254.717,E2 -4254.717} C_VEL
LIN {X 0,Y 531.796,Z 583.825,A -85,B 0,C 180,E1 -4255.435,E2 -4255.435} C_VEL
LIN {X 0,Y 532.023,Z 574.119,A -85,B 0,C 180,E1 -4256.068,E2 -4256.068} C_VEL
LIN {X 0,Y 532.184,Z 563.395,A -85,B 0,C 180,E1 -4256.627,E2 -4256.627} C_VEL
LIN {X 0,Y 531.021,Z 558.342,A -85,B 0,C 180,E1 -4256.901,E2 -4256.901} C_VEL
LIN {X 0,Y 530.995,Z 558.346,A -85,B 0,C 180,E1 -4259.321,E2 -4259.321} C_VEL
LIN {X 0,Y 530.975,Z 558.346,A -85,B 0,C 180,E1 -4262.102,E2 -4262.102} C_VEL
LIN {X 0,Y 530.977,Z 558.346,A -85,B 0,C 180,E1 -4264.853,E2 -4264.853} C_VEL
LIN {X 0,Y 530.961,Z 558.35,A -85,B 0,C 180,E1 -4267.507,E2 -4267.507} C_VEL
LIN {X 0,Y 531.085,Z 558.335,A -85,B 0,C 180,E1 -4270.885,E2 -4270.885} C_VEL
LIN {X 0,Y 531.285,Z 563.864,A -85,B 0,C 180,E1 -4272.869,E2 -4272.869} C_VEL
LIN {X 0,Y 531.248,Z 571.397,A -85,B 0,C 180,E1 -4275.591,E2 -4275.591} C_VEL
LIN {X 0,Y 531.199,Z 579.751,A -85,B 0,C 180,E1 -4278.584,E2 -4278.584} C_VEL
LIN {X 0,Y 531.09,Z 587.532,A -85,B 0,C 180,E1 -4281.328,E2 -4281.328} C_VEL
LIN {X 0,Y 531.023,Z 594.539,A -85,B 0,C 180,E1 -4283.834,E2 -4283.834} C_VEL
LIN {X 0,Y 530.925,Z 601.969,A -85,B 0,C 180,E1 -4286.504,E2 -4286.504} C_VEL
LIN {X 0,Y 530.777,Z 609.811,A -85,B 0,C 180,E1 -4289.389,E2 -4289.389} C_VEL
LIN {X 0,Y 530.678,Z 618.225,A -85,B 0,C 180,E1 -4292.386,E2 -4292.386} C_VEL
LIN {X 0,Y 530.631,Z 621.487,A -85,B 0,C 180,E1 -4293.526,E2 -4293.526} C_VEL
LIN {X 0,Y 532.307,Z 631.947,A -85,B 0,C 180,E1 -4293.804,E2 -4293.804} C_VEL
LIN {X 0,Y 532.145,Z 641.389,A -85,B 0,C 180,E1 -4294.094,E2 -4294.094} C_VEL
LIN {X 0,Y 531.924,Z 651.726,A -85,B 0,C 180,E1 -4294.518,E2 -4294.518} C_VEL
LIN {X 0,Y 531.689,Z 662.367,A -85,B 0,C 180,E1 -4295.082,E2 -4295.082} C_VEL
LIN {X 0,Y 531.502,Z 671.738,A -85,B 0,C 180,E1 -4295.697,E2 -4295.697} C_VEL
LIN {X 0,Y 531.288,Z 680.739,A -85,B 0,C 180,E1 -4296.413,E2 -4296.413} C_VEL
LIN {X 0,Y 531.128,Z 687.322,A -85,B 0,C 180,E1 -4297.024,E2 -4297.024} C_VEL
LIN {X 0,Y 530.944,Z 695.34,A -85,B 0,C 180,E1 -4297.904,E2 -4297.904} C_VEL
LIN {X 0,Y 530.778,Z 702.541,A -85,B 0,C 180,E1 -4298.85,E2 -4298.85} C_VEL
LIN {X 0,Y 530.64,Z 708.915,A -85,B 0,C 180,E1 -4299.858,E2 -4299.858} C_VEL
LIN {X 0,Y 530.606,Z 713.221,A -85,B 0,C 180,E1 -4300.663,E2 -4300.663} C_VEL
LIN {X 0,Y 530.526,Z 718.409,A -85,B 0,C 180,E1 -4301.862,E2 -4301.862} C_VEL
LIN {X 0,Y 530.48,Z 720.836,A -85,B 0,C 180,E1 -4302.528,E2 -4302.528} C_VEL
LIN {X 0,Y 530.374,Z 724.42,A -85,B 0,C 180,E1 -4303.843,E2 -4303.843} C_VEL
LIN {X 0,Y 530.346,Z 725.984,A -85,B 0,C 180,E1 -4304.631,E2 -4304.631} C_VEL
LIN {X 0,Y 530.393,Z 727.709,A -85,B 0,C 180,E1 -4306.202,E2 -4306.202} C_VEL
LIN {X 0,Y 530.359,Z 727.993,A -85,B 0,C 180,E1 -4306.981,E2 -4306.981} C_VEL
LIN {X 0,Y 530.48,Z 727.079,A -85,B 0,C 180,E1 -4308.626,E2 -4308.626} C_VEL
LIN {X 0,Y 530.437,Z 726.231,A -85,B 0,C 180,E1 -4309.31,E2 -4309.31} C_VEL
LIN {X 0,Y 530.43,Z 722.891,A -85,B 0,C 180,E1 -4310.852,E2 -4310.852} C_VEL
LIN {X 0,Y 530.54,Z 719.238,A -85,B 0,C 180,E1 -4312.005,E2 -4312.005} C_VEL
LIN {X 0,Y 530.559,Z 714.499,A -85,B 0,C 180,E1 -4313.153,E2 -4313.153} C_VEL
LIN {X 0,Y 530.677,Z 709.61,A -85,B 0,C 180,E1 -4314.109,E2 -4314.109} C_VEL
LIN {X 0,Y 530.721,Z 703.757,A -85,B 0,C 180,E1 -4315.062,E2 -4315.062} C_VEL
LIN {X 0,Y 530.866,Z 696.736,A -85,B 0,C 180,E1 -4316.015,E2 -4316.015} C_VEL
LIN {X 0,Y 531.034,Z 690.119,A -85,B 0,C 180,E1 -4316.776,E2 -4316.776} C_VEL
LIN {X 0,Y 531.266,Z 681.271,A -85,B 0,C 180,E1 -4317.631,E2 -4317.631} C_VEL
LIN {X 0,Y 531.438,Z 673.078,A -85,B 0,C 180,E1 -4318.295,E2 -4318.295} C_VEL
LIN {X 0,Y 531.634,Z 664.754,A -85,B 0,C 180,E1 -4318.864,E2 -4318.864} C_VEL
LIN {X 0,Y 531.875,Z 654.574,A -85,B 0,C 180,E1 -4319.432,E2 -4319.432} C_VEL
LIN {X 0,Y 532.094,Z 644.995,A -85,B 0,C 180,E1 -4319.858,E2 -4319.858} C_VEL
LIN {X 0,Y 532.251,Z 634.576,A -85,B 0,C 180,E1 -4320.213,E2 -4320.213} C_VEL
LIN {X 0,Y 531.935,Z 628.945,A -85,B 0,C 180,E1 -4320.379,E2 -4320.379} C_VEL
LIN {X 0,Y 530.68,Z 621.486,A -85,B 0,C 180,E1 -4320.569,E2 -4320.569} C_VEL
LIN {X 0,Y 530.755,Z 613.411,A -85,B 0,C 180,E1 -4323.416,E2 -4323.416} C_VEL
LIN {X 0,Y 530.847,Z 607.172,A -85,B 0,C 180,E1 -4325.699,E2 -4325.699} C_VEL
LIN {X 0,Y 530.988,Z 598.892,A -85,B 0,C 180,E1 -4328.755,E2 -4328.755} C_VEL
LIN {X 0,Y 531.086,Z 590.501,A -85,B 0,C 180,E1 -4331.695,E2 -4331.695} C_VEL
LIN {X 0,Y 531.119,Z 582.079,A -85,B 0,C 180,E1 -4334.562,E2 -4334.562} C_VEL
LIN {X 0,Y 531.118,Z 573.714,A -85,B 0,C 180,E1 -4337.306,E2 -4337.306} C_VEL
LIN {X 0,Y 530.991,Z 565.113,A -85,B 0,C 180,E1 -4339.997,E2 -4339.997} C_VEL
LIN {X 0,Y 530.945,Z 558.353,A -85,B 0,C 180,E1 -4342.052,E2 -4342.052} C_VEL
LIN {X 0,Y 531.002,Z 558.347,A -85,B 0,C 180,E1 -4345.058,E2 -4345.058} C_VEL
